ELSIF stRunPara.iPumpType=RudongPump_PumpType.V THEN
	stModbusAddress.iPumpType_Address:=1000;
	stModbusAddress.iHosePipeType_Address:=1001;	
	stModbusAddress.iFluVolumeSet_Address:=1015;
	stModbusAddress.iRuntimeSet_Address:=1018;
	stModbusAddress.iIntervalTime_Address:=1021;
	stModbusAddress.iCycleNumber_Address:=1023;
	stModbusAddress.iBackAngle_Address:=1007;
	stModbusAddress.iMoveDirection_Address:=1009;
	stModbusAddress.iStartStop_Address:=1008;
	stModbusAddress.iFullSpeedStartStop_Address:=1010;
	stModbusAddress.iModuleAddress_Address:=0;//等于0表示不写入
	stModbusAddress.iModuleStartStop_Address:=2003;
	stModbusAddress.iModuleRealFluVolumeSet_Address:=2004;
	stModbusAddress.iRecoveryCalCoefficient_Address:=2006;

	
	
END_IF
END_ACTION

ACTION ACT_PumpPar:
//
(*************************检测配置参数是否匹配成功*********************************)
IF stRunPara.iPumpType=RudongPump_PumpType.DFPluse THEN
	//MiniPump泵头
	IF  stRunPara.iPumpTypeSet=RudongPump_PumpHeadType.MiniPump01 THEN
		st_IOData.O_PumpType:=0;//泵头值为0
			IF stRunPara.iHosePipeTypeSet=RudongPump_SoftPipeType.P13 THEN//13#软管
				st_IOData.O_HosePipeType:=13;//软管类型值13
				IF rFluVolumeSet*1000/135<0.1 THEN
					iMinRunTime:=	0.1;
				ELSE
					iMinRunTime:=	(rFluVolumeSet*1000/135)*0.2+iMinRunTime;
				END_IF
				iMaxRunTime:=	rFluVolumeSet/0.45;//最大流量(0.45微升/秒,0.0024ml/min)	
			ELSIF stRunPara.iHosePipeTypeSet=RudongPump_SoftPipeType.P14 THEN//14#软管
				st_IOData.O_HosePipeType:=14;
				IF rFluVolumeSet*1000/570<0.1 THEN
					iMinRunTime:=	0.1;
				ELSE
					iMinRunTime:=	rFluVolumeSet*1000/135;
				END_IF
				iMaxRunTime:=	(rFluVolumeSet/1.9)*0.2+iMinRunTime;	
			ELSIF stRunPara.iHosePipeTypeSet=RudongPump_SoftPipeType.P19 THEN//19#软管
				st_IOData.O_HosePipeType:=19;
				IF rFluVolumeSet*1000/1240<0.1 THEN
					iMinRunTime:=	0.1;
				ELSE
					iMinRunTime:=	rFluVolumeSet*1000/1240;
				END_IF
				iMaxRunTime:=	(rFluVolumeSet*1000/4.13)*0.1+iMinRunTime;		
			ELSIF stRunPara.iHosePipeTypeSet=RudongPump_SoftPipeType.P16 THEN//16#软管
				st_IOData.O_HosePipeType:=16;
				IF rFluVolumeSet*1000/1880<0.1 THEN
					iMinRunTime:=	0.1;
				ELSE
					iMinRunTime:=	rFluVolumeSet*1000/1880;
				END_IF
				iMaxRunTime:=	(rFluVolumeSet*1000/6.28)*0.2+iMinRunTime;	
			ELSIF stRunPara.iHosePipeTypeSet=RudongPump_SoftPipeType.P25 THEN//25#软管
				st_IOData.O_HosePipeType:=25;
				IF rFluVolumeSet*1000/3100<0.1 THEN
					iMinRunTime:=	0.1;
				ELSE
					iMinRunTime:=	rFluVolumeSet*1000/3100;
				END_IF
				iMaxRunTime:=	(rFluVolumeSet*1000/10.33)*0.2+iMinRunTime;			
		ELSE
				eERRORID:=RudongPump_ERROR.FLT_CONFIGURE_PARA;		
		END_IF
	//UD15
	ELSIF  stRunPara.iPumpTypeSet=RudongPump_PumpHeadType.UD15 THEN
		st_IOData.O_PumpType:=1;//泵头值为0
			IF stRunPara.iHosePipeTypeSet=RudongPump_SoftPipeType.P16 THEN//16#软管
				st_IOData.O_HosePipeType:=16;
				IF rFluVolumeSet*1000/4000<0.1 THEN
					iMinRunTime:=	0.1;
				ELSE
					iMinRunTime:=	rFluVolumeSet*1000/4000;
				END_IF
				iMaxRunTime:=	(rFluVolumeSet*1000/13.33)*0.2+iMinRunTime;		
			ELSIF stRunPara.iHosePipeTypeSet=RudongPump_SoftPipeType.P17 THEN//17#软管
				st_IOData.O_HosePipeType:=17;
				IF rFluVolumeSet*1000/15000<0.1 THEN
					iMinRunTime:=	0.1;
				ELSE
					iMinRunTime:=	rFluVolumeSet*1000/15000;
				END_IF
				iMaxRunTime:=	(rFluVolumeSet*1000/50)*0.2+iMinRunTime;	
			ELSIF stRunPara.iHosePipeTypeSet=RudongPump_SoftPipeType.P25 THEN//25#软管
				st_IOData.O_HosePipeType:=25;
				IF rFluVolumeSet*1000/8000<0.1 THEN
					iMinRunTime:=	0.1;
				ELSE
					iMinRunTime:=	rFluVolumeSet*1000/8000;
				END_IF
				iMaxRunTime:=	(rFluVolumeSet*1000/26.66)*0.2+iMinRunTime;			
		ELSE
				eERRORID:=RudongPump_ERROR.FLT_CONFIGURE_PARA;		
		END_IF

	END_IF
ELSE
		eERRORID:=RudongPump_ERROR.FLT_CONFIGURE_PARA;
END_IF


(*
//MiniPump01泵头
IF  stRunPara.iPumpTypeSet=RudongPump_PumpHeadType.MiniPump01 THEN
		IF stRunPara.iHosePipeTypeSet=RudongPump_SoftPipeType.P13 THEN//13#软管
			iMinRunTime:=	(rFluVolumeSet/8)*60;//最大流量(135微升/秒,8.28ml/min)
			iMaxRunTime:=	(rFluVolumeSet/0.45)*60;//最大流量(0.45微升/秒,0.0024ml/min)	
		ELSIF stRunPara.iHosePipeTypeSet=RudongPump_SoftPipeType.P14 THEN//14#软管
			iMinRunTime:=	(rFluVolumeSet/33)*60;
			iMaxRunTime:=	(rFluVolumeSet/1.9)*60;
		ELSIF stRunPara.iHosePipeTypeSet=RudongPump_SoftPipeType.P19 THEN//19#软管
			iMinRunTime:=	(rFluVolumeSet/77)*60;
			iMaxRunTime:=	(rFluVolumeSet/4.13)*60;	
		ELSIF stRunPara.iHosePipeTypeSet=RudongPump_SoftPipeType.P16 THEN//16#软管
			iMinRunTime:=	(rFluVolumeSet/114)*60;
			iMaxRunTime:=	(rFluVolumeSet/6.28)*60;	
		ELSIF stRunPara.iHosePipeTypeSet=RudongPump_SoftPipeType.P25 THEN//25#软管
			iMinRunTime:=	(rFluVolumeSet/190)*60;
			iMaxRunTime:=	(rFluVolumeSet/10.33)*60;		
		ELSIF stRunPara.iHosePipeTypeSet=RudongPump_SoftPipeType.P1_1 THEN//1x1#软管
			iMinRunTime:=	(rFluVolumeSet/15)*60;
			iMaxRunTime:=	(rFluVolumeSet/4.5)*60;	
		ELSIF stRunPara.iHosePipeTypeSet=RudongPump_SoftPipeType.P2_1 THEN//2x1#软管
			iMinRunTime:=	(rFluVolumeSet/54)*60;
			iMaxRunTime:=	(rFluVolumeSet/4.5)*60;		
		ELSIF stRunPara.iHosePipeTypeSet=RudongPump_SoftPipeType.P2_5_1 THEN//2.5x1#软管
			iMinRunTime:=	(rFluVolumeSet/76)*60;
			iMaxRunTime:=	(rFluVolumeSet/5)*60;		
		ELSIF stRunPara.iHosePipeTypeSet=RudongPump_SoftPipeType.P3_1 THEN//3x1#软管
			iMinRunTime:=	(rFluVolumeSet/108)*60;
			iMaxRunTime:=	(rFluVolumeSet/5)*60;
	ELSE
			eERRORID:=RudongPump_ERROR.FLT_CONFIGURE_PARA;		
	END_IF		
	
//MiniPump02泵头
ELSIF  stRunPara.iPumpTypeSet=RudongPump_PumpHeadType.MiniPump02 THEN
	IF stRunPara.iHosePipeTypeSet=RudongPump_SoftPipeType.P1_1 THEN//1x1#软管
		iMinRunTime:=	(rFluVolumeSet/15.01)*60;
		iMaxRunTime:=	(rFluVolumeSet/0.005)*60;	
	ELSIF stRunPara.iHosePipeTypeSet=RudongPump_SoftPipeType.P2_1 THEN//2x1#软管
		iMinRunTime:=	(rFluVolumeSet/54.63)*60;
		iMaxRunTime:=	(rFluVolumeSet/0.018)*60;		
	ELSIF stRunPara.iHosePipeTypeSet=RudongPump_SoftPipeType.P2_5_1 THEN//2.5x1#软管
		iMinRunTime:=	(rFluVolumeSet/76.84)*60;
		iMaxRunTime:=	(rFluVolumeSet/0.0256)*60;
	ELSE
			eERRORID:=RudongPump_ERROR.FLT_CONFIGURE_PARA;						
	END_IF	

//HandyPump01泵头
ELSIF  stRunPara.iPumpTypeSet=RudongPump_PumpHeadType.HandyPump01 THEN
	IF stRunPara.iHosePipeTypeSet=RudongPump_SoftPipeType.P13 THEN//13#软管,三滚轮
		iMinRunTime:=	(rFluVolumeSet/10)*60;
		iMaxRunTime:=	(rFluVolumeSet/0.0033)*60;	
	ELSIF stRunPara.iHosePipeTypeSet=RudongPump_SoftPipeType.P14 THEN//14#软管,三滚轮
		iMinRunTime:=	(rFluVolumeSet/56)*60;
		iMaxRunTime:=	(rFluVolumeSet/0.0187)*60;		
	ELSIF stRunPara.iHosePipeTypeSet=RudongPump_SoftPipeType.P19 THEN//19#软管,三滚轮
		iMinRunTime:=	(rFluVolumeSet/111)*60;
		iMaxRunTime:=	(rFluVolumeSet/0.0371)*60;
	ELSIF stRunPara.iHosePipeTypeSet=RudongPump_SoftPipeType.P16 THEN//16#软管,三滚轮
		iMinRunTime:=	(rFluVolumeSet/190)*60;
		iMaxRunTime:=	(rFluVolumeSet/0.0636)*60;		
	ELSIF stRunPara.iHosePipeTypeSet=RudongPump_SoftPipeType.P25 THEN//25#软管,三滚轮
		iMinRunTime:=	(rFluVolumeSet/365)*60;
		iMaxRunTime:=	(rFluVolumeSet/0.1219)*60;
	ELSE
			eERRORID:=RudongPump_ERROR.FLT_CONFIGURE_PARA;						
	END_IF

//HandyPump02泵头
ELSIF  stRunPara.iPumpTypeSet=RudongPump_PumpHeadType.HandyPump02 THEN
	IF stRunPara.iHosePipeTypeSet=RudongPump_SoftPipeType.P13 THEN//13#软管,三滚轮
		iMinRunTime:=	(rFluVolumeSet/10)*60;
		iMaxRunTime:=	(rFluVolumeSet/0.0033)*60;	
	ELSIF stRunPara.iHosePipeTypeSet=RudongPump_SoftPipeType.P14 THEN//14#软管,三滚轮
		iMinRunTime:=	(rFluVolumeSet/56)*60;
		iMaxRunTime:=	(rFluVolumeSet/0.0187)*60;		
	ELSIF stRunPara.iHosePipeTypeSet=RudongPump_SoftPipeType.P19 THEN//19#软管,三滚轮
		iMinRunTime:=	(rFluVolumeSet/111)*60;
		iMaxRunTime:=	(rFluVolumeSet/0.0371)*60;
	ELSIF stRunPara.iHosePipeTypeSet=RudongPump_SoftPipeType.P16 THEN//16#软管,三滚轮
		iMinRunTime:=	(rFluVolumeSet/190)*60;
		iMaxRunTime:=	(rFluVolumeSet/0.0636)*60;	
	ELSE
			eERRORID:=RudongPump_ERROR.FLT_CONFIGURE_PARA;							
	END_IF

//EasyPumpI_III泵头,单通道
ELSIF  stRunPara.iPumpTypeSet=RudongPump_PumpHeadType.EasyPumpI_III THEN
	IF stRunPara.iHosePipeTypeSet=RudongPump_SoftPipeType.P13 THEN//13#软管
		iMinRunTime:=	(rFluVolumeSet/32)*60;
		iMaxRunTime:=	(rFluVolumeSet/0.0053)*60;	
	ELSIF stRunPara.iHosePipeTypeSet=RudongPump_SoftPipeType.P14 THEN//14#软管
		iMinRunTime:=	(rFluVolumeSet/162)*60;
		iMaxRunTime:=	(rFluVolumeSet/0.027)*60;		
	ELSIF stRunPara.iHosePipeTypeSet=RudongPump_SoftPipeType.P19 THEN//19#软管
		iMinRunTime:=	(rFluVolumeSet/330)*60;
		iMaxRunTime:=	(rFluVolumeSet/0.055)*60;
	ELSIF stRunPara.iHosePipeTypeSet=RudongPump_SoftPipeType.P16 THEN//16#软管
		iMinRunTime:=	(rFluVolumeSet/560)*60;
		iMaxRunTime:=	(rFluVolumeSet/0.093)*60;	
	ELSIF stRunPara.iHosePipeTypeSet=RudongPump_SoftPipeType.P25 THEN//25#软管
		iMinRunTime:=	(rFluVolumeSet/1180)*60;
		iMaxRunTime:=	(rFluVolumeSet/0.197)*60;	
	ELSIF stRunPara.iHosePipeTypeSet=RudongPump_SoftPipeType.P17 THEN//17#软管
		iMinRunTime:=	(rFluVolumeSet/2000)*60;
		iMaxRunTime:=	(rFluVolumeSet/0.333)*60;	
	ELSIF stRunPara.iHosePipeTypeSet=RudongPump_SoftPipeType.P18 THEN//18#软管
		iMinRunTime:=	(rFluVolumeSet/2580)*60;
		iMaxRunTime:=	(rFluVolumeSet/0.430)*60;	
	ELSE
			eERRORID:=RudongPump_ERROR.FLT_CONFIGURE_PARA;							
	END_IF

//EasyPumpII_IV泵头,单通道
ELSIF  stRunPara.iPumpTypeSet=RudongPump_PumpHeadType.EasyPumpII_IV THEN
	IF stRunPara.iHosePipeTypeSet=RudongPump_SoftPipeType.P15 THEN//15#软管
		iMinRunTime:=	(rFluVolumeSet/1080)*60;
		iMaxRunTime:=	(rFluVolumeSet/0.0180)*60;	
	ELSIF stRunPara.iHosePipeTypeSet=RudongPump_SoftPipeType.P24 THEN//24#软管
		iMinRunTime:=	(rFluVolumeSet/1640)*60;
		iMaxRunTime:=	(rFluVolumeSet/0.273)*60;		
	ELSIF stRunPara.iHosePipeTypeSet=RudongPump_SoftPipeType.P35 THEN//35#软管
		iMinRunTime:=	(rFluVolumeSet/2300)*60;
		iMaxRunTime:=	(rFluVolumeSet/0.383)*60;
	ELSIF stRunPara.iHosePipeTypeSet=RudongPump_SoftPipeType.P36 THEN//36#软管
		iMinRunTime:=	(rFluVolumeSet/3100)*60;
		iMaxRunTime:=	(rFluVolumeSet/0.517)*60;	
	ELSE
			eERRORID:=RudongPump_ERROR.FLT_CONFIGURE_PARA;							
	END_IF

//EasyPumpV_VI泵头,双通道
ELSIF  stRunPara.iPumpTypeSet=RudongPump_PumpHeadType.EasyPumpV_VI THEN
		IF stRunPara.iHosePipeTypeSet=RudongPump_SoftPipeType.P13 THEN//13#软管
		iMinRunTime:=	(rFluVolumeSet/32)*60;
		iMaxRunTime:=	(rFluVolumeSet/0.0053)*60;	
	ELSIF stRunPara.iHosePipeTypeSet=RudongPump_SoftPipeType.P14 THEN//14#软管
		iMinRunTime:=	(rFluVolumeSet/162)*60;
		iMaxRunTime:=	(rFluVolumeSet/0.0027)*60;		
	ELSIF stRunPara.iHosePipeTypeSet=RudongPump_SoftPipeType.P19 THEN//19#软管
		iMinRunTime:=	(rFluVolumeSet/330)*60;
		iMaxRunTime:=	(rFluVolumeSet/0.0055)*60;
	ELSIF stRunPara.iHosePipeTypeSet=RudongPump_SoftPipeType.P16 THEN//16#软管
		iMinRunTime:=	(rFluVolumeSet/560)*60;
		iMaxRunTime:=	(rFluVolumeSet/0.093)*60;		
	ELSIF stRunPara.iHosePipeTypeSet=RudongPump_SoftPipeType.P25 THEN//25#软管
		iMinRunTime:=	(rFluVolumeSet/1180)*60;
		iMaxRunTime:=	(rFluVolumeSet/0.197)*60;
	ELSE
			eERRORID:=RudongPump_ERROR.FLT_CONFIGURE_PARA;							
	END_IF
	
END_IF


END_IF

*)
		


//参数超出范围报错	
IF rFluVolumeSet<>0 THEN
	IF rRuntimeSet<iMinRunTime OR rRuntimeSet>iMaxRunTime OR  iMaxRunTime<iMinRunTime THEN
		eERRORID:=RudongPump_ERROR.FLT_CONFIGURE_PARA;
	END_IF
END_IF
END_ACTION

ACTION ACTMap:
ACT_GetModbusAddress();
_fResetCheck(CLK:=xResetRequest);
xRdyCmd := eState = STATE.DORMANT AND eERRORID = RudongPump_ERROR.No_ERROR;//检测是否允许指令控制(初始状态，没有报警发生)
xDone:=_xDone AND xExecute;
xError:=eState=STATE.INERROR;//报错发生
(**********************************检测是否有模式切换********************************)
_rManual(CLK:=xAutoMode);
_fManual(CLK:=xAutoMode);
IF eState <> STATE.DORMANT//只有在运行的时候，才会检测是否有模式切换发生
THEN
	IF _rManual.Q OR _fManual.Q
	THEN
		_xModeChange := TRUE;//通知系统有模式切换发生
	END_IF	
END_IF
IF eState = STATE.DORMANT//要是待机模式下，切换模式，是不会起作用的
THEN
	_xModeChange := FALSE;
END_IF


////
//调用MODBUS TCP功能
_fbModbusTCP.stSysPar.sRemoteHost:=stPara.strSlaveIP;//'192.168.1.20';
_fbModbusTCP.stSysPar.nRemotePort:=stPara.nRemotePort;
_fbModbusTCP.stSysPar.xSlaveAdr:=stPara.bySlaveID;
_fbModbusTCP(
	stParIn:= , 
	stSysPar:= , 
	xResetRequest:=xResetRequest , 
	stOpera:= , 
	xDone=> , 
	xBusy=> , 
	xError=> , 
	eERRORID=> , 
	eTCPErrorID=> , 	
	sModbusError=> , 
	xRdyCmd=> , 
	sError=> , 
	stParOut=> );
END_ACTION

METHOD PROTECTED CmdCalParWrite
VAR_OUTPUT
	xComplete: BOOL;
END_VAR
// return the real actual fault number
IF eERRORID <> RudongPump_ERROR.No_ERROR
THEN
  RETURN;  
END_IF

CASE _diCmdState OF	

	0://清空缓冲区
		SysMemSet(ADR(_fbModbusTCP.stParIn.aSendBuffer),0,SIZEOF(_fbModbusTCP.stParIn.aSendBuffer));		
		IF _fbModbusTCP.xRdyCmd THEN
			_diCmdState:=_diCmdState+1;
		ELSE
			eERRORID:=RudongPump_ERROR.FLT_Mobdus;
			_diCmdState:=999;
		END_IF
		
	1://单元实际液量设定
		_fbModbusTCP.stParIn.iHoldingRegisterAddress:=stModbusAddress.iModuleRealFluVolumeSet_Address;
		_fbModbusTCP.stParIn.iHoldingRegisterNum:=2;	
		_pDataControl:=ADR(iModuleRealVolume);	
 		_fbModbusTCP.stParIn.aSendBuffer[1]:=	_pDataControl[3];
 		_fbModbusTCP.stParIn.aSendBuffer[2]:=	_pDataControl[2];		
 		_fbModbusTCP.stParIn.aSendBuffer[3]:=	_pDataControl[1];		
 		_fbModbusTCP.stParIn.aSendBuffer[4]:=	_pDataControl[0];		
		_fbModbusTCP.stOpera.xSetMultiHoldingRegister:=TRUE;
		IF _fbModbusTCP.xDone THEN
			_fbModbusTCP.xExecute:=FALSE;
			_diCmdState:=_diCmdState+1;
		END_IF
		IF _fbModbusTCP.xError THEN
			eERRORID:=RudongPump_ERROR.FLT_Mobdus;
			_diCmdState:=999;
		END_IF
		
	2://
		xComplete := TRUE; 
		
	ELSE
		;	
END_CASE
END_METHOD

METHOD PROTECTED CmdCalReset
VAR_OUTPUT
	xComplete: BOOL;
END_VAR
// return the real actual fault number
IF eERRORID <> RudongPump_ERROR.No_ERROR
THEN
  RETURN;  
END_IF

CASE _diCmdState OF	
		
	0://清空缓冲区
		SysMemSet(ADR(_fbModbusTCP.stParIn.aSendBuffer),0,SIZEOF(_fbModbusTCP.stParIn.aSendBuffer));		
		IF _fbModbusTCP.xRdyCmd THEN
			_diCmdState:=_diCmdState+1;
		ELSE
			eERRORID:=RudongPump_ERROR.FLT_Mobdus;
			_diCmdState:=999;
		END_IF
		
	1://发送灌装系数复位指令
 		_fbModbusTCP.stParIn.aSendBuffer[1]:=16#00;
 		_fbModbusTCP.stParIn.aSendBuffer[2]:=16#01;		
		_fbModbusTCP.stParIn.iHoldingRegisterAddress:=stModbusAddress.iRecoveryCalCoefficient_Address;
		_fbModbusTCP.stParIn.iHoldingRegisterNum:=1;		 	
		_fbModbusTCP.stOpera.xSetSingalHoldingRegister:=TRUE;
		IF _fbModbusTCP.xDone THEN
			_fbModbusTCP.xExecute:=FALSE;
			_diCmdState:=_diCmdState+1;
		END_IF
		IF _fbModbusTCP.xError THEN
			eERRORID:=RudongPump_ERROR.FLT_Mobdus;
			_diCmdState:=999;
		END_IF

	2://
		xComplete := TRUE; 
		
	ELSE
		;	
END_CASE
END_METHOD

METHOD PROTECTED CmdPumpCal
VAR_OUTPUT
	xComplete: BOOL;
END_VAR
// return the real actual fault number
IF eERRORID <> RudongPump_ERROR.No_ERROR
THEN
  RETURN;  
END_IF

CASE _diCmdState OF	
	0://清空缓冲区
		SysMemSet(ADR(_fbModbusTCP.stParIn.aSendBuffer),0,SIZEOF(_fbModbusTCP.stParIn.aSendBuffer));		
		IF _fbModbusTCP.xRdyCmd THEN
			_diCmdState:=_diCmdState+1;
		ELSE
			eERRORID:=RudongPump_ERROR.FLT_Mobdus;
			_diCmdState:=999;
		END_IF
	
	 1://发送灌装液量,1002,REAL
		_fbModbusTCP.stParIn.iHoldingRegisterAddress:=stModbusAddress.iFluVolumeSet_Address;
		_fbModbusTCP.stParIn.iHoldingRegisterNum:=2;	
		_pDataControl:=ADR(rFluVolumeSet);	
 		_fbModbusTCP.stParIn.aSendBuffer[1]:=	_pDataControl[3];
 		_fbModbusTCP.stParIn.aSendBuffer[2]:=	_pDataControl[2];		
 		_fbModbusTCP.stParIn.aSendBuffer[3]:=	_pDataControl[1];		
 		_fbModbusTCP.stParIn.aSendBuffer[4]:=	_pDataControl[0];		
		_fbModbusTCP.stOpera.xSetMultiHoldingRegister:=TRUE;
		IF _fbModbusTCP.xDone THEN
			_fbModbusTCP.xExecute:=FALSE;
			_diCmdState:=_diCmdState+1;
		END_IF
		IF _fbModbusTCP.xError THEN
			eERRORID:=RudongPump_ERROR.FLT_Mobdus;
			_diCmdState:=999;
		END_IF		
	
	 2://发送灌装时间,1004,REAL
		_fbModbusTCP.stParIn.iHoldingRegisterAddress:=stModbusAddress.iRuntimeSet_Address;
		_fbModbusTCP.stParIn.iHoldingRegisterNum:=2;
		rRuntimeSet			:=stRunPara.rCalTime;
		_pDataControl:=ADR(rRuntimeSet);	
 		_fbModbusTCP.stParIn.aSendBuffer[1]:=	_pDataControl[3];
 		_fbModbusTCP.stParIn.aSendBuffer[2]:=	_pDataControl[2];		
 		_fbModbusTCP.stParIn.aSendBuffer[3]:=	_pDataControl[1];		
 		_fbModbusTCP.stParIn.aSendBuffer[4]:=	_pDataControl[0];		
		_fbModbusTCP.stOpera.xSetMultiHoldingRegister:=TRUE;
		IF _fbModbusTCP.xDone THEN
			_fbModbusTCP.xExecute:=FALSE;
			_diCmdState:=_diCmdState+1;
		END_IF
		IF _fbModbusTCP.xError THEN
			eERRORID:=RudongPump_ERROR.FLT_Mobdus;
			_diCmdState:=999;
		END_IF

	 3://发送灌装方向,1010,UINT
		IF eCmd = RudongPump_CMD.Cmd_Push OR eCmd = RudongPump_CMD.Cmd_CalPump
		THEN
			_fbModbusTCP.stParIn.aSendBuffer[1]:=16#00;
			_fbModbusTCP.stParIn.aSendBuffer[2]:=16#01;		
		END_IF
		IF eCmd = RudongPump_CMD.Cmd_Pull 
		THEN
			_fbModbusTCP.stParIn.aSendBuffer[1]:=16#00;
			_fbModbusTCP.stParIn.aSendBuffer[2]:=16#00;			
		END_IF		
		_fbModbusTCP.stParIn.iHoldingRegisterAddress:=stModbusAddress.iMoveDirection_Address;
		_fbModbusTCP.stParIn.iHoldingRegisterNum:=1;			 	
		_fbModbusTCP.stOpera.xSetSingalHoldingRegister:=TRUE;
		IF _fbModbusTCP.xDone THEN
			_fbModbusTCP.xExecute:=FALSE;
			_diCmdState:=_diCmdState+1;
		END_IF
		IF _fbModbusTCP.xError THEN
			eERRORID:=RudongPump_ERROR.FLT_Mobdus;
			_diCmdState:=999;
		END_IF		

	4://发送重复次数,1008,UINT
		_pDataControl:=ADR(iCycleNumber);	
 		_fbModbusTCP.stParIn.aSendBuffer[1]:=_pDataControl[1];
 		_fbModbusTCP.stParIn.aSendBuffer[2]:=_pDataControl[0];		
		_fbModbusTCP.stParIn.iHoldingRegisterAddress:=stModbusAddress.iCycleNumber_Address;
		_fbModbusTCP.stParIn.iHoldingRegisterNum:=1;		 	
		_fbModbusTCP.stOpera.xSetSingalHoldingRegister:=TRUE;
		IF _fbModbusTCP.xDone THEN
			_fbModbusTCP.xExecute:=FALSE;
			_diCmdState:=_diCmdState+1;
		END_IF
		IF _fbModbusTCP.xError THEN
			eERRORID:=RudongPump_ERROR.FLT_Mobdus;
			_diCmdState:=999;
		END_IF	
		
	5://单元地址设定,2000,UINT
		_pDataControl:=ADR(iModuleAdress);	
 		_fbModbusTCP.stParIn.aSendBuffer[1]:=_pDataControl[1];
 		_fbModbusTCP.stParIn.aSendBuffer[2]:=_pDataControl[0];		
		_fbModbusTCP.stParIn.iHoldingRegisterAddress:=stModbusAddress.iModuleAddress_Address;
		_fbModbusTCP.stParIn.iHoldingRegisterNum:=1;		
		IF  _fbModbusTCP.stParIn.iHoldingRegisterAddress<>0 THEN	
			_fbModbusTCP.stOpera.xSetSingalHoldingRegister:=TRUE;
			IF _fbModbusTCP.xDone THEN
				_fbModbusTCP.xExecute:=FALSE;
				_diCmdState:=_diCmdState+1;
			END_IF
			IF _fbModbusTCP.xError THEN
				eERRORID:=RudongPump_ERROR.FLT_Mobdus;
				_diCmdState:=999;
			END_IF
		ELSE
			_diCmdState:=_diCmdState+1;//地址为0 则跳过设置
		END_IF
		
	6://灌装启动,2003,UINT	
 		_fbModbusTCP.stParIn.aSendBuffer[1]:=16#00;
 		_fbModbusTCP.stParIn.aSendBuffer[2]:=16#01;		
		_fbModbusTCP.stParIn.iHoldingRegisterAddress:=stModbusAddress.iModuleStartStop_Address;
		_fbModbusTCP.stParIn.iHoldingRegisterNum:=1;		 	
		_fbModbusTCP.stOpera.xSetSingalHoldingRegister:=TRUE;
		IF _fbModbusTCP.xDone THEN
			_fbModbusTCP.xExecute:=FALSE;
			_diCmdState:=_diCmdState+1;
		END_IF
		IF _fbModbusTCP.xError THEN
			eERRORID:=RudongPump_ERROR.FLT_Mobdus;
			_diCmdState:=999;
		END_IF

	7://查询蠕动泵运行状态,2003,UINT
		_fbModbusTCP.stParIn.iHoldingRegisterAddress:=stModbusAddress.iModuleStartStop_Address;
		_fbModbusTCP.stParIn.iHoldingRegisterNum:=1;		 	
		_fbModbusTCP.stOpera.xReadHoldingRegisters:=TRUE;
		IF _fbModbusTCP.xDone THEN
			_fbModbusTCP.xExecute:=FALSE;
			_diCmdState:=_diCmdState+1;
		END_IF
		IF _fbModbusTCP.xError THEN
			eERRORID:=RudongPump_ERROR.FLT_Mobdus;
			_diCmdState:=999;
		END_IF			
		
	8://判断运行状态,并延时
		IF _fbModbusTCP.stParOut.aRcvBuffer[1]=0 AND _fbModbusTCP.stParOut.aRcvBuffer[2]=0 THEN
			xComplete:=TRUE;
		ELSE
			xRunning:=TRUE;
			_tonDelay(IN:=TRUE,PT:=T#0.5S);
			IF _tonDelay.Q THEN
				_tonDelay(IN:=FALSE);
				_diCmdState:=7;
			END_IF
		END_IF
		
	ELSE
		;	
END_CASE
END_METHOD

METHOD PROTECTED CmdRunAction
VAR_OUTPUT
	xComplete: BOOL;
END_VAR
// return the real actual fault number
IF eERRORID <> RudongPump_ERROR.No_ERROR
THEN
  RETURN;  
END_IF

CASE _diCmdState OF	
	0://清空缓冲区
		SysMemSet(ADR(_fbModbusTCP.stParIn.aSendBuffer),0,SIZEOF(_fbModbusTCP.stParIn.aSendBuffer));		
		IF _fbModbusTCP.xRdyCmd THEN
			IF xNeedConfigurePara THEN
				_diCmdState:=_diCmdState+1;
			ELSE
				_diCmdState:=6;//如果不需要配置则直接启动
			END_IF			
		ELSE
			eERRORID:=RudongPump_ERROR.FLT_Mobdus;
			_diCmdState:=999;
		END_IF

	 1://发送虚假灌装时间,1004,REAL
		_fbModbusTCP.stParIn.iHoldingRegisterAddress:=stModbusAddress.iRuntimeSet_Address;
		_fbModbusTCP.stParIn.iHoldingRegisterNum:=2;
		_pDataControl:=ADR(iMaxRunTime);	
 		_fbModbusTCP.stParIn.aSendBuffer[1]:=	_pDataControl[3];
 		_fbModbusTCP.stParIn.aSendBuffer[2]:=	_pDataControl[2];		
 		_fbModbusTCP.stParIn.aSendBuffer[3]:=	_pDataControl[1];		
 		_fbModbusTCP.stParIn.aSendBuffer[4]:=	_pDataControl[0];		
		_fbModbusTCP.stOpera.xSetMultiHoldingRegister:=TRUE;
		IF _fbModbusTCP.xDone THEN
			_fbModbusTCP.xExecute:=FALSE;
			_diCmdState:=_diCmdState+1;
		END_IF
		IF _fbModbusTCP.xError THEN
			eERRORID:=RudongPump_ERROR.FLT_Mobdus;
			_diCmdState:=999;
		END_IF		
		
	 2://发送灌装液量,1002,REAL
		_fbModbusTCP.stParIn.iHoldingRegisterAddress:=stModbusAddress.iFluVolumeSet_Address;
		_fbModbusTCP.stParIn.iHoldingRegisterNum:=2;	
		_pDataControl:=ADR(rFluVolumeSet);	
 		_fbModbusTCP.stParIn.aSendBuffer[1]:=	_pDataControl[3];
 		_fbModbusTCP.stParIn.aSendBuffer[2]:=	_pDataControl[2];		
 		_fbModbusTCP.stParIn.aSendBuffer[3]:=	_pDataControl[1];		
 		_fbModbusTCP.stParIn.aSendBuffer[4]:=	_pDataControl[0];		
		_fbModbusTCP.stOpera.xSetMultiHoldingRegister:=TRUE;
		IF _fbModbusTCP.xDone THEN
			_fbModbusTCP.xExecute:=FALSE;
			_diCmdState:=_diCmdState+1;
		END_IF
		IF _fbModbusTCP.xError THEN
			eERRORID:=RudongPump_ERROR.FLT_Mobdus;
			_diCmdState:=999;
		END_IF			

	 3://发送实际灌装时间,1004,REAL
		_fbModbusTCP.stParIn.iHoldingRegisterAddress:=stModbusAddress.iRuntimeSet_Address;
		_fbModbusTCP.stParIn.iHoldingRegisterNum:=2;
		_pDataControl:=ADR(rRuntimeSet);	
 		_fbModbusTCP.stParIn.aSendBuffer[1]:=	_pDataControl[3];
 		_fbModbusTCP.stParIn.aSendBuffer[2]:=	_pDataControl[2];		
 		_fbModbusTCP.stParIn.aSendBuffer[3]:=	_pDataControl[1];		
 		_fbModbusTCP.stParIn.aSendBuffer[4]:=	_pDataControl[0];		
		_fbModbusTCP.stOpera.xSetMultiHoldingRegister:=TRUE;
		IF _fbModbusTCP.xDone THEN
			_fbModbusTCP.xExecute:=FALSE;
			_diCmdState:=_diCmdState+1;
		END_IF
		IF _fbModbusTCP.xError THEN
			eERRORID:=RudongPump_ERROR.FLT_Mobdus;
			_diCmdState:=999;
		END_IF
		
	 4://发送灌装方向,1010,UINT
		IF eCmd = RudongPump_CMD.Cmd_Push
		THEN
			_fbModbusTCP.stParIn.aSendBuffer[1]:=16#00;
			_fbModbusTCP.stParIn.aSendBuffer[2]:=16#01;		
		END_IF
		IF eCmd = RudongPump_CMD.Cmd_Pull 
		THEN
			_fbModbusTCP.stParIn.aSendBuffer[1]:=16#00;
			_fbModbusTCP.stParIn.aSendBuffer[2]:=16#00;			
		END_IF		
		_fbModbusTCP.stParIn.iHoldingRegisterAddress:=stModbusAddress.iMoveDirection_Address;
		_fbModbusTCP.stParIn.iHoldingRegisterNum:=1;			 	
		_fbModbusTCP.stOpera.xSetSingalHoldingRegister:=TRUE;
		IF _fbModbusTCP.xDone THEN
			_fbModbusTCP.xExecute:=FALSE;
			_diCmdState:=_diCmdState+1;
		END_IF
		IF _fbModbusTCP.xError THEN
			eERRORID:=RudongPump_ERROR.FLT_Mobdus;
			_diCmdState:=999;
		END_IF		

	5://发送重复次数,1008,UINT
		_pDataControl:=ADR(iCycleNumber);	
 		_fbModbusTCP.stParIn.aSendBuffer[1]:=_pDataControl[1];
 		_fbModbusTCP.stParIn.aSendBuffer[2]:=_pDataControl[0];		
		_fbModbusTCP.stParIn.iHoldingRegisterAddress:=stModbusAddress.iCycleNumber_Address;
		_fbModbusTCP.stParIn.iHoldingRegisterNum:=1;		 	
		_fbModbusTCP.stOpera.xSetSingalHoldingRegister:=TRUE;
		IF _fbModbusTCP.xDone THEN
			_fbModbusTCP.xExecute:=FALSE;
			_diCmdState:=_diCmdState+1;
		END_IF
		IF _fbModbusTCP.xError THEN
			eERRORID:=RudongPump_ERROR.FLT_Mobdus;
			_diCmdState:=999;
		END_IF

	6://发送启动,1011,UINT
		_fbModbusTCP.stParIn.aSendBuffer[1]:=16#00;
		_fbModbusTCP.stParIn.aSendBuffer[2]:=16#01;	
		_fbModbusTCP.stParIn.iHoldingRegisterAddress:=stModbusAddress.iStartStop_Address;
		_fbModbusTCP.stParIn.iHoldingRegisterNum:=1;		 	
		_fbModbusTCP.stOpera.xSetSingalHoldingRegister:=TRUE;
		IF _fbModbusTCP.xDone THEN
			_fbModbusTCP.xExecute:=FALSE;
			_diCmdState:=_diCmdState+1;
		END_IF
		IF _fbModbusTCP.xError THEN
			eERRORID:=RudongPump_ERROR.FLT_Mobdus;
			_diCmdState:=999;
		END_IF
	7://查询蠕动泵运行状态,1011,UINT
		_fbModbusTCP.stParIn.iHoldingRegisterAddress:=stModbusAddress.iStartStop_Address;
		_fbModbusTCP.stParIn.iHoldingRegisterNum:=1;		 	
		_fbModbusTCP.stOpera.xReadHoldingRegisters:=TRUE;
		IF _fbModbusTCP.xDone THEN
			_fbModbusTCP.xExecute:=FALSE;
			_diCmdState:=_diCmdState+1;
		END_IF
		IF _fbModbusTCP.xError THEN
			eERRORID:=RudongPump_ERROR.FLT_Mobdus;
			_diCmdState:=999;
		END_IF			
		
	8://判断运行状态,并延时
		IF _fbModbusTCP.stParOut.aRcvBuffer[1]=0 AND _fbModbusTCP.stParOut.aRcvBuffer[2]=0 THEN
			xComplete:=TRUE;
		ELSE
			xRunning:=TRUE;
			_tonDelay(IN:=TRUE,PT:=T#1S);
			IF _tonDelay.Q THEN
				_tonDelay(IN:=FALSE);
				_diCmdState:=7;
			END_IF
		END_IF
	
	
		
	ELSE
		;	
END_CASE
END_METHOD

METHOD PROTECTED CyclicAction
VAR_OUTPUT
	xComplete: BOOL;
END_VAR
IF xAbort=0 THEN
    IF xFirstInvocation THEN
    (*
    * Staring
    * for then first (!) invocaion,
    * sample then input variables
    *)			
    _diCmdState:= 0;
		_iNGCount := 0;
		_iActRunNumber := 0;
		xFirstInvocation:=0;			
    END_IF    
    REPEAT 				
		  (**************************检查是否有硬件报错(检测总线是否报错)**********************************) 
			IF _xConnectError
			THEN
				eERRORID := RudongPump_ERROR.FLT_CONNECT;//子站通讯报警
			END_IF
		
	
			//检测停止指令是否发生
			_rStopCmdTrig(CLK:= NOT xEStop OR (stDeviceOpe.xStop_Hmi AND NOT xAutoMode AND NOT xDeviceRunning) OR (stDeviceOpe.xStop_Auto AND (xAutoMode OR xDeviceRunning))
													OR (stDeviceOpe.xFullSpeedStop_Hmi AND NOT xAutoMode AND NOT xDeviceRunning) OR (stDeviceOpe.xFullSpeedStop_Auto AND (xAutoMode OR xDeviceRunning)));		
		  IF _rStopCmdTrig.Q//检测到停止指令
			THEN
				_diCmdState := 0;
				eCmd := RudongPump_CMD.Cmd_Stop;
				_tonCmdTimeout(in:=FALSE);
				_tonDelay(IN:= FALSE);
				_tonTimeout(in:=FALSE);
			END_IF
			
			ACT_PumpPar();//检查参数	
			
			
			CASE eCmd OF//判断指令类型
				RudongPump_CMD.Cmd_Pull,RudongPump_CMD.Cmd_Push://执行夹爪指令(夹紧和松开指令)
					CmdRunAction(xComplete=> xComplete);	
							
				RudongPump_CMD.Cmd_Stop,RudongPump_CMD.Cmd_FullSpeedStop://执行过程中等待停止指令(分为运行停止和全速停止)
					mCmdStopAction(xComplete=> xComplete);
					
				RudongPump_CMD.Cmd_Configure://(用于配置参数)
					mCmdConfigureAction(xComplete=> xComplete);
					
				RudongPump_CMD.Cmd_FullSpeedPush,RudongPump_CMD.Cmd_FullSpeedPull://全速启动控制（用于清洗和充满试管）
					mCmdFullSpeedStartAction(xComplete=> xComplete);
					
				RudongPump_CMD.Cmd_CalPump:
					CmdPumpCal(xComplete=> xComplete);

				RudongPump_CMD.Cmd_CalReset:
					CmdCalReset(xComplete=> xComplete);		

				RudongPump_CMD.Cmd_CalParWrite:
					CmdCalParWrite(xComplete=> xComplete);		
				ELSE
					;	
				END_CASE		   
      UNTIL (TRUE)
	END_REPEAT
END_IF

IF xAbort OR xComplete OR eERRORID<>RudongPump_ERROR.No_ERROR THEN    
    (*
    * Cleaning
    * => free as much allocated resources as possible
    *)    
    tOperationTimer(IN:=0);
END_IF
END_METHOD

METHOD PRIVATE FINAL HandleAbortedState
VAR_INPUT
END_VAR
VAR_OUTPUT
	xAgain: BOOL;
END_VAR
VAR
	xComplete: BOOL;
END_VAR
IF xAborted AND xResetRequest THEN
    eState:=STATE.RESETING;
    xAgain:=1;
ELSE
    xBusy:=0;
    xAborted:=1;
    //xResetRequest:=(xExecute=0);
    xAgain:=0;(* !!! *)
END_IF
END_METHOD

METHOD PRIVATE FINAL HandleAbortingState
VAR_INPUT
END_VAR
VAR_OUTPUT
	xAgain: BOOL;
END_VAR
VAR
	xComplete: BOOL;
END_VAR
AbortAction(xComplete=> xComplete, eERRORID=> eERRORID);

IF eERRORID<>RudongPump_ERROR.No_ERROR THEN
    eState:=STATE.INERROR;
    xAgain:=1;
ELSIF xComplete THEN
    eState:=STATE.ABORTED;
    xAgain:=1;
END_IF
END_METHOD

METHOD PRIVATE FINAL HandleDoneState
VAR_INPUT
END_VAR
VAR_OUTPUT
	xAgain: BOOL;
END_VAR
//在运行过程中要是切换模式，再运行完成之后，检测到模式的切换，就需要回到初始位置，进行下一次执行准备
IF _xDone AND ((xExecute=0) OR ( _xModeChange AND NOT _xAutoOpe)  OR ( NOT xAutoMode AND NOT xDeviceRunning AND ( NOT _xAutoOpe OR _xHMIOpe))) THEN
	eState:=STATE.RESETING;
	xAgain:=1;
ELSE
	xBusy:=0;
	_xDone:=1;
	xAgain:=0;(* !!! *)
END_IF
END_METHOD

METHOD PRIVATE FINAL HandleDormantState
VAR_INPUT
END_VAR
VAR_OUTPUT
	xAgain: BOOL;
END_VAR
IF xExecute THEN
    xBusy:=1;
    eState:=STATE.EXECUTING;
    xAgain:=1;
END_IF
//下面两个报警一旦报警就需要发生
IF _xConnectError 
THEN//出现这个进行报警
	eERRORID := RudongPump_ERROR.FLT_CONNECT;//子站通讯报警
END_IF

IF _fResetCheck.Q//清空报警
THEN
	eERRORID := RudongPump_ERROR.No_ERROR;
END_IF
IF  xAutoMode OR xDeviceRunning THEN
	xAutomodeFlag:=TRUE;
ELSE
	xAutomodeFlag:=FALSE;
END_IF


IF eErrorID = RudongPump_ERROR.NO_ERROR 
THEN
	IF   xRunILC   THEN
		FOR k:=1 TO 5 BY 1 DO
			//PULL
			_rOperaTrig[k](CLK:=xRunILC AND (stDeviceOpe.xPull_Hmi[k] AND NOT xAutomodeFlag) OR (stDeviceOpe.xPull_Auto[k] AND xAutomodeFlag));
			IF _rOperaTrig[k].Q //
			THEN
				rFluVolumeSet	:=stRunPara.rPullFluVolume[k];
				rRuntimeSet		:=stRunPara.rPullRuntime[k];
				iCycleNumber	:=stRunPara.iPullCycleNumber[k];
				eCmd 			:= RudongPump_CMD.Cmd_Pull;
				xExecute		:= TRUE;
			END_IF		
			//PUSH
			_rOperaTrig[k+5](CLK:=xRunILC AND (stDeviceOpe.xPush_Hmi[k] AND NOT xAutomodeFlag) OR (stDeviceOpe.xPush_Auto[k] AND xAutomodeFlag));
			IF _rOperaTrig[k+5].Q 
			THEN
				rFluVolumeSet	:=stRunPara.rPushFluVolume[k];  
				rRuntimeSet		:=stRunPara.rPushRuntime[k];    
				iCycleNumber	:=stRunPara.iPushCycleNumber[k];
				eCmd 			:= RudongPump_CMD.Cmd_Push;
				xExecute 		:= TRUE;
			END_IF				
		END_FOR
		//STOP
		 IF(stDeviceOpe.xStop_Hmi AND  NOT xAutomodeFlag) OR NOT xEStop OR stDeviceOpe.xStop_Auto    THEN
				eCmd := RudongPump_CMD.Cmd_Stop;
				xExecute := TRUE;
		 END_IF
		//FullSpeedPull
		IF (stDeviceOpe.xFullSpeedPull_Hmi AND  NOT xAutomodeFlag) OR (stDeviceOpe.xFullSpeedPull_Auto AND  xAutomodeFlag) THEN
			eCmd := RudongPump_CMD.Cmd_FullSpeedPull;
			xExecute := TRUE;
		END_IF
		//FullSpeedPush
		IF (stDeviceOpe.xFullSpeedPush_Hmi AND NOT xAutomodeFlag ) OR (stDeviceOpe.xFullSpeedPush_Auto AND xAutomodeFlag) THEN	
			eCmd := RudongPump_CMD.Cmd_FullSpeedPush;
			xExecute := TRUE;
		END_IF
		//FullSpeedStop
		 IF (stDeviceOpe.xFullSpeedStop_Hmi AND NOT xAutomodeFlag) OR (stDeviceOpe.xFullSpeedStop_Auto AND xAutomodeFlag) THEN	
			eCmd := RudongPump_CMD.Cmd_FullSpeedStop;
			xExecute := TRUE;
		END_IF
		//Configure
		IF (stDeviceOpe.xConfigure_Hmi AND NOT xAutomodeFlag) OR (stDeviceOpe.xConfigure_Auto AND xAutomodeFlag) THEN	
			eCmd := RudongPump_CMD.Cmd_Configure;
			xExecute := TRUE;
		END_IF
		
	END_IF		
		//校准
		IF stDeviceOpe.xPumpCal_Hmi OR stDeviceOpe.xPumpCal_Auto THEN
			rFluVolumeSet		:=stRunPara.rCalFluVolume;
			rRuntimeSet			:=stRunPara.rCalTime;
			iCycleNumber		:=stRunPara.rCalNum;	
			iModuleAdress		:=stRunPara.iModuleAdress;
			iModuleSpeed		:=stRunPara.rModuleSpeed;		
			eCmd 				:= RudongPump_CMD.Cmd_CalPump;
			xExecute 			:= TRUE;		
		END_IF
		
		//复位校准系数为初始值
		IF stDeviceOpe.xResetCalcoeffCal_Hmi THEN	
			eCmd 				:= RudongPump_CMD.Cmd_CalReset;
			xExecute 			:= TRUE;		
		END_IF
	
		//校准参数写入
		IF stDeviceOpe.xCalParWrite_Hmi OR stDeviceOpe.xCalParWrite_Auto THEN	
			eCmd 								:= RudongPump_CMD.Cmd_CalParWrite;
			iModuleRealVolume		:=stRunPara.rModuleRealFluVolume;					
			xExecute 						:= TRUE;		
		END_IF	
			
END_IF
END_METHOD

METHOD PRIVATE FINAL  HandleErrorState
VAR_INPUT
END_VAR
VAR_OUTPUT
	xAgain: BOOL;
END_VAR
IF xRudongPump_ERROR AND  (xResetRequest OR NOT xExecute) THEN
    eState:=STATE.RESETING;
    xAgain:=1;
ELSE
    xBusy:=0;
    xRudongPump_ERROR:=1;    
    xAgain:=0;(* !!! *)
END_IF
END_METHOD

METHOD PRIVATE FINAL HandleExecutingState
VAR_INPUT
END_VAR
VAR_OUTPUT
	xAgain: BOOL;
END_VAR
VAR
	xComplete: BOOL;
END_VAR
IF xAbort=0 THEN   
    CyclicAction(xComplete=> xComplete);
END_IF

IF eERRORID<>RudongPump_ERROR.No_ERROR THEN
    eState:=STATE.INERROR;
    xAgain:=1;
ELSIF xAbort THEN
    eState:=STATE.ABORTING;
    xAgain:=1;
ELSIF xComplete THEN
    eState:=STATE.DONE;
    xAgain:=1;
END_IF
END_METHOD

METHOD PRIVATE FINAL HandleResettingState
VAR_INPUT
END_VAR
VAR_OUTPUT
	xAgain: BOOL;
END_VAR
VAR
	xComplete: BOOL;
END_VAR
ResetAction(xComplete=> xComplete);

IF xComplete THEN
	xExecute:=0;//清除输入指令 
    xBusy:=0;
    _xDone:=0;
    xRudongPump_ERROR:=0;
    xAborted:=0;
    eERRORID:=RudongPump_ERROR.No_ERROR;
    eState:=STATE.DORMANT;
    xFirstInvocation:=1;
    xAgain:=0;(* !!! *)
END_IF
END_METHOD

METHOD PROTECTED mCmdConfigureAction
VAR_OUTPUT
	xComplete: BOOL;
END_VAR
// return the real actual fault number
IF eERRORID <> RudongPump_ERROR.No_ERROR
THEN
  RETURN;  
END_IF

CASE _diCmdState OF

	0://清空缓冲区
		SysMemSet(ADR(_fbModbusTCP.stParIn.aSendBuffer),0,SIZEOF(_fbModbusTCP.stParIn.aSendBuffer));		
		IF _fbModbusTCP.xRdyCmd THEN
			_diCmdState:=_diCmdState+1;
		ELSE
			eERRORID:=RudongPump_ERROR.FLT_Mobdus;
			_diCmdState:=999;
		END_IF
		
	 1://发送泵头编号,1000,UINT
		_pDataControl:=ADR(st_IOData.O_PumpType);	
 		_fbModbusTCP.stParIn.aSendBuffer[1]:=_pDataControl[1];
 		_fbModbusTCP.stParIn.aSendBuffer[2]:=_pDataControl[0];		
		_fbModbusTCP.stParIn.iHoldingRegisterAddress:=stModbusAddress.iPumpType_Address;
		_fbModbusTCP.stParIn.iHoldingRegisterNum:=1;		 	
		_fbModbusTCP.stOpera.xSetSingalHoldingRegister:=TRUE;
		IF _fbModbusTCP.xDone THEN
			_fbModbusTCP.xExecute:=FALSE;
			_diCmdState:=_diCmdState+1;
		END_IF
		IF _fbModbusTCP.xError THEN
			eERRORID:=RudongPump_ERROR.FLT_Mobdus;
			_diCmdState:=999;
		END_IF

	 2://发送软管编号,1001,UINT
		_pDataControl:=ADR(st_IOData.O_HosePipeType);	
 		_fbModbusTCP.stParIn.aSendBuffer[1]:=_pDataControl[1];
 		_fbModbusTCP.stParIn.aSendBuffer[2]:=_pDataControl[0];		
		_fbModbusTCP.stParIn.iHoldingRegisterAddress:=stModbusAddress.iHosePipeType_Address;
		_fbModbusTCP.stParIn.iHoldingRegisterNum:=1;		 	
		_fbModbusTCP.stOpera.xSetSingalHoldingRegister:=TRUE;
		IF _fbModbusTCP.xDone THEN
			_fbModbusTCP.xExecute:=FALSE;
			_diCmdState:=_diCmdState+1;
		END_IF
		IF _fbModbusTCP.xError THEN
			eERRORID:=RudongPump_ERROR.FLT_Mobdus;
			_diCmdState:=999;
		END_IF

	3://
		xComplete:=TRUE;
















	ELSE
		;
END_CASE
END_METHOD

METHOD PROTECTED mCmdFullSpeedStartAction
VAR_OUTPUT
	xComplete: BOOL;
END_VAR
// return the real actual fault number
IF eERRORID <> RudongPump_ERROR.No_ERROR
THEN
  RETURN;  
END_IF

CASE _diCmdState OF
	0://清空缓冲区
		SysMemSet(ADR(_fbModbusTCP.stParIn.aSendBuffer),0,SIZEOF(_fbModbusTCP.stParIn.aSendBuffer));		
		IF _fbModbusTCP.xRdyCmd THEN
			_diCmdState:=_diCmdState+1;
		ELSE
			eERRORID:=RudongPump_ERROR.FLT_Mobdus;
			_diCmdState:=999;
		END_IF

	 1://发送灌装方向,1010,UINT
		IF eCmd = RudongPump_CMD.Cmd_FullSpeedPush
		THEN
			_fbModbusTCP.stParIn.aSendBuffer[1]:=16#00;
			_fbModbusTCP.stParIn.aSendBuffer[2]:=16#01;		
		END_IF
		IF eCmd = RudongPump_CMD.Cmd_FullSpeedPull 
		THEN
			_fbModbusTCP.stParIn.aSendBuffer[1]:=16#00;
			_fbModbusTCP.stParIn.aSendBuffer[2]:=16#00;			
		END_IF		
		_fbModbusTCP.stParIn.iHoldingRegisterAddress:=stModbusAddress.iMoveDirection_Address;
		_fbModbusTCP.stParIn.iHoldingRegisterNum:=1;			 	
		_fbModbusTCP.stOpera.xSetSingalHoldingRegister:=TRUE;
		IF _fbModbusTCP.xDone THEN
			_fbModbusTCP.xExecute:=FALSE;
			_diCmdState:=_diCmdState+1;
		END_IF
		IF _fbModbusTCP.xError THEN
			eERRORID:=RudongPump_ERROR.FLT_Mobdus;
			_diCmdState:=999;
		END_IF	
		
	2://发送启动,1012,UINT
		_fbModbusTCP.stParIn.aSendBuffer[1]:=16#00;
		_fbModbusTCP.stParIn.aSendBuffer[2]:=16#01;	
		_fbModbusTCP.stParIn.iHoldingRegisterAddress:=stModbusAddress.iFullSpeedStartStop_Address;
		_fbModbusTCP.stParIn.iHoldingRegisterNum:=1;		 	
		_fbModbusTCP.stOpera.xSetSingalHoldingRegister:=TRUE;
		IF _fbModbusTCP.xDone THEN
			_fbModbusTCP.xExecute:=FALSE;
			_diCmdState:=_diCmdState+1;
		END_IF
		IF _fbModbusTCP.xError THEN
			eERRORID:=RudongPump_ERROR.FLT_Mobdus;
			_diCmdState:=999;
		END_IF
		
	3://查询蠕动泵运行状态,1012,UINT
		_fbModbusTCP.stParIn.iHoldingRegisterAddress:=stModbusAddress.iStartStop_Address;
		_fbModbusTCP.stParIn.iHoldingRegisterNum:=1;		 	
		_fbModbusTCP.stOpera.xReadHoldingRegisters:=TRUE;
		IF _fbModbusTCP.xDone THEN
			_fbModbusTCP.xExecute:=FALSE;
			_diCmdState:=_diCmdState+1;
		END_IF
		IF _fbModbusTCP.xError THEN
			eERRORID:=RudongPump_ERROR.FLT_Mobdus;
			_diCmdState:=999;
		END_IF			
		
	4://判断运行状态,并延时
		IF _fbModbusTCP.stParOut.aRcvBuffer[1]<>0 OR _fbModbusTCP.stParOut.aRcvBuffer[2]<>0 THEN
			xRunning:=TRUE;
			xComplete:=TRUE;
		ELSE
			_tonDelay(IN:=TRUE,PT:=T#0.5S);
			IF _tonDelay.Q THEN
				_tonDelay(IN:=FALSE);
				_diCmdState:=2;
			END_IF
		END_IF		
		
		
	ELSE
		;
END_CASE
END_METHOD

METHOD PROTECTED mCmdStopAction
VAR_OUTPUT
	xComplete: BOOL;
END_VAR
// return the real actual fault number
IF eERRORID <> RudongPump_ERROR.No_ERROR
THEN
  RETURN;  
END_IF

CASE _diCmdState OF
	0://清空缓冲区
		_tonDelay(IN:=_fbModbusTCP.xRdyCmd,PT:=T#100MS);
		SysMemSet(ADR(_fbModbusTCP.stParIn.aSendBuffer),0,SIZEOF(_fbModbusTCP.stParIn.aSendBuffer));		
		IF _fbModbusTCP.xRdyCmd AND _tonDelay.Q THEN
			_diCmdState:=_diCmdState+1;
		ELSE
			_fbModbusTCP.xExecute:=FALSE;
		END_IF

	1://发送启动停止,1012,UINT
		_fbModbusTCP.stParIn.aSendBuffer[1]:=16#00;
		_fbModbusTCP.stParIn.aSendBuffer[2]:=16#00;	
		_fbModbusTCP.stParIn.iHoldingRegisterAddress:=stModbusAddress.iFullSpeedStartStop_Address;
		_fbModbusTCP.stParIn.iHoldingRegisterNum:=1;		 	
		_fbModbusTCP.stOpera.xSetSingalHoldingRegister:=TRUE;
		IF _fbModbusTCP.xDone THEN
			_fbModbusTCP.xExecute:=FALSE;
			_diCmdState:=_diCmdState+1;
		END_IF
		IF _fbModbusTCP.xError THEN
			eERRORID:=RudongPump_ERROR.FLT_Mobdus;
			_diCmdState:=999;
		END_IF		
 		
	2://发送启动停止,1011,UINT
		_fbModbusTCP.stParIn.aSendBuffer[1]:=16#00;
		_fbModbusTCP.stParIn.aSendBuffer[2]:=16#00;	
		_fbModbusTCP.stParIn.iHoldingRegisterAddress:=stModbusAddress.iStartStop_Address;
		_fbModbusTCP.stParIn.iHoldingRegisterNum:=1;		 	
		_fbModbusTCP.stOpera.xSetSingalHoldingRegister:=TRUE;
		IF _fbModbusTCP.xDone THEN
			_fbModbusTCP.xExecute:=FALSE;
			_diCmdState:=_diCmdState+1;
		END_IF
		IF _fbModbusTCP.xError THEN
			eERRORID:=RudongPump_ERROR.FLT_Mobdus;
			_diCmdState:=999;
		END_IF	
 		
	3://发送启动停止,2003,UINT
		_fbModbusTCP.stParIn.aSendBuffer[1]:=16#00;
		_fbModbusTCP.stParIn.aSendBuffer[2]:=16#00;	
		_fbModbusTCP.stParIn.iHoldingRegisterAddress:=stModbusAddress.iModuleStartStop_Address;
		_fbModbusTCP.stParIn.iHoldingRegisterNum:=1;		 	
		_fbModbusTCP.stOpera.xSetSingalHoldingRegister:=TRUE;
		IF _fbModbusTCP.xDone THEN
			_fbModbusTCP.xExecute:=FALSE;
			_diCmdState:=_diCmdState+1;
		END_IF
		IF _fbModbusTCP.xError THEN
			eERRORID:=RudongPump_ERROR.FLT_Mobdus;
			_diCmdState:=999;
		END_IF	

	4://完成	
		xComplete:=TRUE;
		
	ELSE
		;
END_CASE
END_METHOD

METHOD PROTECTED ResetAction
VAR_OUTPUT
	xComplete: BOOL;
END_VAR
(*
* Cleaning
* => free all allocated resources
* => reinitialize instance variables
*)
tOperationTimer(IN:=0);
tInvocationTimer(IN:=0);
xRunning:=FALSE;
// init command state
//xExecute:=FALSE;
_diCmdState := 0;
_tonCmdTimeout(in:=FALSE);
_tonDelay(IN:= FALSE);
_tonTimeout(in:=FALSE);
_xModeChange := FALSE;
_rStopCmdTrig(CLK:=FALSE);
_iNGCount := 0;
_fbModbusTCP.xExecute:=FALSE;
FOR k:=1 TO 15 BY 1 DO
	_rOperaTrig[k](CLK:=FALSE);
END_FOR	
	
stDeviceOpe.xConfigure_Auto:= stDeviceOpe.xConfigure_Hmi:= FALSE;
stDeviceOpe.xStop_Auto:= stDeviceOpe.xStop_Hmi:= FALSE;
stDeviceOpe.xFullSpeedPull_Auto:= stDeviceOpe.xFullSpeedPull_Hmi:= FALSE;
stDeviceOpe.xFullSpeedPush_Auto:= stDeviceOpe.xFullSpeedPush_Hmi:= FALSE;
stDeviceOpe.xFullSpeedStop_Auto:= stDeviceOpe.xFullSpeedStop_Hmi:= FALSE;
FOR k:=1 TO 5 DO
	stDeviceOpe.xPull_Auto[k]:= stDeviceOpe.xPull_Hmi[k] := FALSE;
	stDeviceOpe.xPush_Auto[k]:= stDeviceOpe.xPush_Hmi[k] := FALSE;
END_FOR

stDeviceOpe.xPumpCal_Auto:=stDeviceOpe.xPumpCal_Hmi:=FALSE;
stDeviceOpe.xCalParWrite_Auto:=stDeviceOpe.xCalParWrite_Hmi:=FALSE;
stDeviceOpe.xResetCalcoeffCal_Hmi:=FALSE;
xResetRequest:=FALSE;
//复位完成
xComplete:=1;
END_METHOD

END_FUNCTION_BLOCK

// ---- POUs/003_FB/53_RudongPump/41 Modbus指令/FB_ModbusTCP.TcPOU
FUNCTION_BLOCK FB_ModbusTCP
VAR_INPUT
	///参数输入	
	stParIn: ModbusParIn;
	///系统参数输入
	stSysPar: Modbus_SysPar;
	///复位操作
	xResetRequest: BOOL;
	///操作
	stOpera: Modbus_Operation;
	///指令执行
	{attribute 'hide' := ''}
	xExecute: BOOL;
END_VAR
VAR_OUTPUT
	///完成条件满足
	xDone: BOOL;
	///动作正在执行
	xBusy: BOOL;
	///错误条件满足
	xError: BOOL;
	eERRORID: Modbus_ErrorCode;
	eTCPErrorID: UDINT;
	///MODBUS错误码
	sModbusError: STRING;
	///指令被打断，一般是处于急停中
	xAborted: BOOL;
	///代表指令准备完成
	xRdyCmd: BOOL;
	///用于显示的错误代码
	sError: STRING;
	///参数输出
	stParOut: ModbusParOut;
END_VAR
VAR
	///MODBUS TCP收发序列号
	{attribute 'hide' := ''}
	iModbusTCP_ComID: WORD;
	///指令中断
	{attribute 'hide' := ''}
	xAbort: BOOL;
	///接收缓存区域(byte数组)
	{attribute 'hide' := ''}
	_rxBuffer: ARRAY[1..MAX_PLCPRJ_RXBUFFER_SIZE] OF BYTE;
	///执行指令
	{attribute 'hide' := ''}
	eCmd: Modbus_Cmd;
	{attribute 'hide' := ''}
	i: INT;
	{attribute 'hide' := ''}
	j: INT;
	{attribute 'hide' := ''}
	k: INT;
	{attribute 'hide' := ''}
	xOpe: BOOL;
	{attribute 'hide' := ''}
	_diCmdState: DINT;
	{attribute 'hide' := ''}
	_diReadParStep: DINT;
	{attribute 'hide' := ''}
	_fbTcpIpClient: FB_TcpIpClient;
	///当前状态
	{attribute 'hide' := ''}
	eState: STATE;
	{attribute 'hide' := ''}
	xFirstInvocation: BOOL := TRUE;
	{attribute 'hide' := ''}
	xTimeOut: BOOL;
	{attribute 'hide' := ''}
	tOperationTimer: TON;
	{attribute 'hide' := ''}
	_tDelay: TON;
	{attribute 'hide' := ''}
	_twaitDelay: TON;
	{attribute 'hide' := ''}
	_first: BOOL;
	///发送NG计数	
	{attribute 'hide' := ''}
	_iSendNGCount: INT;
	{attribute 'hide' := ''}
	_tonCmdTimeout: TON;
	{attribute 'hide' := ''}
	_tonDelay: TON;
	{attribute 'hide' := ''}
	_tonTimeout: TON;
	{attribute 'hide' := ''}
	_xDone: BOOL;
END_VAR
VAR_TEMP
	xAgain: BOOL;
END_VAR

IF NOT _first 
THEN
	_first := TRUE;
ELSE
	_fbTcpIpClient.nRemotePort := stSysPar.nRemotePort;
	_fbTcpIpClient.sRemoteHost := stSysPar.sRemoteHost;
	xAgain:=0;
	_fbTcpIpClient();
	eTCPErrorID := _fbTcpIpClient.udiErrorID;
	xRdyCmd := ( eState = STATE.DORMANT );
	xDone := _xDone AND xExecute;//判断是否处于当前流程的Done状态
	REPEAT
		CASE eState OF
			STATE.DORMANT:
				HandleDormantState(xAgain=> xAgain);
			STATE.EXECUTING:
				HandleExecutingState(xAgain=> xAgain);
			STATE.DONE:
				HandleDoneState(xAgain=> xAgain);
			STATE.INERROR:
				HandleErrorState(xAgain=> xAgain);
			STATE.ABORTING:
				HandleAbortingState(xAgain=> xAgain);
			STATE.ABORTED:
				HandleAbortedState(xAgain=> xAgain);
			STATE.RESETING:
				HandleResettingState(xAgain=> xAgain);
			END_CASE
	UNTIL (xAgain=0)
	END_REPEAT
END_IF


xOpe:=
stOpera.xReadCoilStatus OR 
stOpera.xReadHoldingRegisters OR 
stOpera.xReadInputRegisters OR 
stOpera.xReadInputStatus OR 
stOpera.xSetMultiCoil OR 
stOpera.xSetMultiHoldingRegister OR 
stOpera.xSetSingalCoil OR 
stOpera.xSetSingalHoldingRegister;

//错误码
CASE eERRORID OF
	Modbus_ErrorCode.FLT_CMD						:	sError:='FLT_CMD';
	Modbus_ErrorCode.FLT_CMDTIMEOUT			:	sError:='FLT_CMDTIMEOUT';
	Modbus_ErrorCode.FLT_MODBUS_ERROR		:	sError:=sModbusError;
	Modbus_ErrorCode.FLT_NoResponse			:	sError:='FLT_NoResponse';
	Modbus_ErrorCode.FLT_PAROVERFLOW		:	sError:='FLT_PAROVERFLOW';	
	Modbus_ErrorCode.FLT_RECEIVE_ERROR	:	sError:='FLT_RECEIVE_ERROR';	
	Modbus_ErrorCode.FLT_SEND_ERROR			:	sError:='FLT_SEND_ERROR';	
	Modbus_ErrorCode.No_ERROR						:	sError:='No_ERROR';	
END_CASE

{attribute 'hide' := ''}
METHOD PROTECTED AbortAction
VAR_OUTPUT
	xComplete: BOOL;
END_VAR
(*
* Cleaning
* => abort all running operation
* => if an NBS.ERROR codition is reached, set eErrorID to a Value rather then NBS.ERROR.NO_ERROR 
*)
xComplete:=1;
eErrorID:=Modbus_ErrorCode.NO_ERROR;
END_METHOD

METHOD Cmd_ReadCoil
VAR_OUTPUT
	xComplete: BOOL;
END_VAR
IF eERRORID <> Modbus_ErrorCode.No_ERROR
THEN
  RETURN;  
END_IF

CASE _diCmdState OF	
	0://清空数据
		_fbTcpIpClient.xEnable := FALSE;	
		_tonDelay(IN:= TRUE,pt:=T#1MS);
		_tonTimeout(IN:= FALSE);
		SysMemSet( ADR(_fbTcpIpClient.aToServer ), 0, SIZEOF(_fbTcpIpClient.aToServer) );//清除发送区域
		SysMemSet( ADR(_rxBuffer ), 0, SIZEOF(_rxBuffer) );//清除接收报告数据缓存区域
		SysMemSet( ADR(stParOut.aRcvBuffer ), 0, SIZEOF(stParOut.aRcvBuffer) );//清除接收报告数据缓存区域		
		SysMemSet( ADR(stParOut.aRcvCoilBuffer ), 0, SIZEOF(stParOut.aRcvCoilBuffer) );//清除接收报告数据缓存区域		
		_fbTcpIpClient.xNeedReceive := TRUE;//默认都是需要有收发交互的	
		_fbTcpIpClient.xNeedDisConnect := TRUE;//默认都是需要有收发交互的		
		IF _tonDelay.Q THEN
			_tonDelay(IN:= FALSE,pt:=T#20MS);
			_diCmdState:=_diCmdState+1;	
		END_IF	
	
	1://拼接指令
		_fbTcpIpClient.aToServer[1] :=TO_BYTE(SHR(iModbusTCP_ComID,8));
		_fbTcpIpClient.aToServer[2] :=TO_BYTE(iModbusTCP_ComID);
		_fbTcpIpClient.aToServer[3] :=16#00;//		
		_fbTcpIpClient.aToServer[4] :=16#00;//
		_fbTcpIpClient.aToServer[5] :=16#00;//		
		_fbTcpIpClient.aToServer[6] :=16#06;//后面发送字节数量,6个字节			
		_fbTcpIpClient.aToServer[7] :=stSysPar.xSlaveAdr;//设备地址
		_fbTcpIpClient.aToServer[8] :=16#01;//查询功能码01
		_fbTcpIpClient.aToServer[9] :=TO_BYTE(SHR(stParIn.iHoldingRegisterAddress,8));
		_fbTcpIpClient.aToServer[10] :=TO_BYTE(stParIn.iHoldingRegisterAddress);      //读取寄存器起始地址 
		_fbTcpIpClient.aToServer[11] :=TO_BYTE(SHR(stParIn.iCoilNum,8));
		_fbTcpIpClient.aToServer[12] :=TO_BYTE(stParIn.iCoilNum);       		//读取寄存器数量
		_fbTcpIpClient.udiSendNumber:=12;
		IF stParIn.iCoilNum>2000 OR stParIn.iCoilNum<1 THEN
			eERRORID:=Modbus_ErrorCode.FLT_PAROVERFLOW	;//参数超出范围
			_diCmdState := 999;			
		END_IF		
		IF _fbTcpIpClient.xRdyCmd
		THEN
			_diCmdState:=_diCmdState+1;
		ELSE
			_fbTcpIpClient.xEnable := FALSE;
		END_IF
		
	2://接收数据
		_fbTcpIpClient.xEnable 		:= TRUE;	
		IF _fbTcpIpClient.xDone//接收成功
		THEN	
			_iSendNgCount 					:= 0;//代表数据接收成功									
			_rxBuffer 							:= _fbTcpIpClient.rxBuffer;							
			_diCmdState:=_diCmdState+1;			
		END_IF
		//发送出错
		IF _fbTcpIpClient.xError 
		THEN//以太网功能报警，一般就是网络建立有问题，此时一般需要去查网络问题
			_iSendNgCount := _iSendNgCount + 1;
			IF _iSendNgCount <= 3//3次重发
			THEN		
				_tDelay(in:=TRUE,PT:=T#100MS);	
				IF _tDelay.Q
				THEN
					_tDelay(in:=FALSE);
					_diCmdState:=0;//重发
				END_IF							
			ELSE			
				eERRORID:=Modbus_ErrorCode.FLT_SEND_ERROR	;//指令发送出错，可能是通信异常	
				_diCmdState := 999;
			END_IF						
		END_IF			
		
	3://校验MODBUS返回指令
		_tonTimeout(IN:= TRUE,pt:=T#3S);
		IF _tonTimeout.Q THEN
			_tonTimeout(IN:=FALSE);
			eERRORID:=Modbus_ErrorCode.FLT_NoResponse	;//无响应
			_diCmdState := 999;			
		END_IF			
		
	//指令返回OK
		IF 
			_rxBuffer[1]=_fbTcpIpClient.aToServer[1] AND
			_rxBuffer[2]=_fbTcpIpClient.aToServer[2] AND
			_rxBuffer[3]=_fbTcpIpClient.aToServer[3] AND
			_rxBuffer[4]=_fbTcpIpClient.aToServer[4] AND
			_rxBuffer[7]=stSysPar.xSlaveAdr AND
			_rxBuffer[8]=16#01//功能码
		THEN
			IF //如果是8的倍数
				stParIn.iCoilNum MOD 8 =0 AND
				_rxBuffer[5]=TO_BYTE(SHR(stParIn.iCoilNum/8+3,8)) AND
				_rxBuffer[6]=TO_BYTE(stParIn.iCoilNum/8+3) AND
				_rxBuffer[9]=TO_BYTE(stParIn.iCoilNum/8)
			THEN
				_diCmdState:=_diCmdState+1;				
			END_IF	
			IF //如果不是8的倍数
				stParIn.iCoilNum MOD 8 <>0 AND
				_rxBuffer[5]=TO_BYTE(SHR(stParIn.iCoilNum/8+4,8)) AND
				_rxBuffer[6]=TO_BYTE(stParIn.iCoilNum/8+4) AND
				_rxBuffer[9]=TO_BYTE(stParIn.iCoilNum/8+1) 
			THEN
				_diCmdState:=_diCmdState+1;				
			END_IF			
		END_IF
		
		//指令返回MODBUS错误码
		IF 
			_rxBuffer[1]=_fbTcpIpClient.aToServer[1] AND
			_rxBuffer[2]=_fbTcpIpClient.aToServer[2] AND
			_rxBuffer[3]=_fbTcpIpClient.aToServer[3] AND
			_rxBuffer[4]=_fbTcpIpClient.aToServer[4] AND
			_rxBuffer[5]=0 AND 
			_rxBuffer[6]=3 AND
			_rxBuffer[7]=_fbTcpIpClient.aToServer[7] AND
			_rxBuffer[8]=16#81//功能码
		THEN
			sModbusError:=ModbusTCP_ErrorQuery(_rxBuffer[9]);//解析MODBUS错误代码
			eERRORID:=Modbus_ErrorCode.FLT_MODBUS_ERROR	;//Modbus错误
			_diCmdState := 999;				
		END_IF		
		
		//指令返回异常,重发3次
		IF 
			_rxBuffer[1]<>_fbTcpIpClient.aToServer[1] OR
			_rxBuffer[2]<>_fbTcpIpClient.aToServer[2] OR
			_rxBuffer[3]<>0 OR
			_rxBuffer[4]<>0 OR
			_rxBuffer[7]<>_fbTcpIpClient.aToServer[7]
		THEN		
			_iSendNgCount := _iSendNgCount + 1;
			IF _iSendNgCount <= 3//3次重发
			THEN		
				_tDelay(in:=TRUE,PT:=T#100MS);	
				IF _tDelay.Q
				THEN
					_tDelay(in:=FALSE);
					_diCmdState:=0;//重发
				END_IF							
			ELSE	
				eERRORID:=Modbus_ErrorCode.FLT_RECEIVE_ERROR	;//接收指令错误
				_diCmdState := 999;
			END_IF		
		END_IF
		
	4://解析数据
		SysMemCpy(ADR(stparout.aRcvBuffer),ADR(_rxBuffer[10]),TO_INT(_rxBuffer[9]));
		iModbusTCP_ComID:=iModbusTCP_ComID+1;
		_diCmdState:=_diCmdState+1;	
		
	5://获取BOOL数据
		FOR i:=1 TO _rxBuffer[9] BY 1 DO		
			stparout.aRcvCoilBuffer[(i-1)*8+1]	:=stparout.aRcvBuffer[i].00;
			stparout.aRcvCoilBuffer[(i-1)*8+2]	:=stparout.aRcvBuffer[i].01;		
			stparout.aRcvCoilBuffer[(i-1)*8+3]	:=stparout.aRcvBuffer[i].02;
			stparout.aRcvCoilBuffer[(i-1)*8+4]	:=stparout.aRcvBuffer[i].03;
			stparout.aRcvCoilBuffer[(i-1)*8+5]	:=stparout.aRcvBuffer[i].04;
			stparout.aRcvCoilBuffer[(i-1)*8+6]	:=stparout.aRcvBuffer[i].05;
			stparout.aRcvCoilBuffer[(i-1)*8+7]	:=stparout.aRcvBuffer[i].06;
			stparout.aRcvCoilBuffer[(i-1)*8+8]	:=stparout.aRcvBuffer[i].07;
		END_FOR
		xComplete:=TRUE;

END_CASE
END_METHOD

METHOD Cmd_ReadHoldingRegister
VAR_OUTPUT
	xComplete: BOOL;
END_VAR
IF eERRORID <> Modbus_ErrorCode.No_ERROR
THEN
  RETURN;  
END_IF

CASE _diCmdState OF	
	0://清空数据
		_fbTcpIpClient.xEnable := FALSE;	
		_tonDelay(IN:= TRUE,pt:=T#1MS);
		_tonTimeout(IN:= FALSE);
		SysMemSet( ADR(_fbTcpIpClient.aToServer ), 0, SIZEOF(_fbTcpIpClient.aToServer) );//清除发送区域
		SysMemSet( ADR(_rxBuffer ), 0, SIZEOF(_rxBuffer) );//清除接收报告数据缓存区域
		SysMemSet( ADR(stParOut.aRcvBuffer ), 0, SIZEOF(stParOut.aRcvBuffer) );//清除接收报告数据缓存区域		
		SysMemSet( ADR(stParOut.aRcvCoilBuffer ), 0, SIZEOF(stParOut.aRcvCoilBuffer) );//清除接收报告数据缓存区域		
		_fbTcpIpClient.xNeedReceive := TRUE;//默认都是需要有收发交互的	
		_fbTcpIpClient.xNeedDisConnect := TRUE;//默认都是需要有收发交互的		
		IF _tonDelay.Q THEN
			_tonDelay(IN:= FALSE,pt:=T#20MS);
			_diCmdState:=_diCmdState+1;	
		END_IF	
	
	1://拼接指令
		_fbTcpIpClient.aToServer[1] :=TO_BYTE(SHR(iModbusTCP_ComID,8));
		_fbTcpIpClient.aToServer[2] :=TO_BYTE(iModbusTCP_ComID);
		_fbTcpIpClient.aToServer[3] :=16#00;//		
		_fbTcpIpClient.aToServer[4] :=16#00;//
		_fbTcpIpClient.aToServer[5] :=16#00;//		
		_fbTcpIpClient.aToServer[6] :=16#06;//后面发送字节数量,6个字节			
		_fbTcpIpClient.aToServer[7] :=stSysPar.xSlaveAdr;//设备地址
		_fbTcpIpClient.aToServer[8] :=16#03;//查询功能码03
		_fbTcpIpClient.aToServer[9] :=TO_BYTE(SHR(stParIn.iHoldingRegisterAddress,8));
		_fbTcpIpClient.aToServer[10] :=TO_BYTE(stParIn.iHoldingRegisterAddress);      //读取寄存器起始地址 
		_fbTcpIpClient.aToServer[11] :=TO_BYTE(SHR(stParIn.iHoldingRegisterNum,8));
		_fbTcpIpClient.aToServer[12] :=TO_BYTE(stParIn.iHoldingRegisterNum);       		//读取寄存器数量
		_fbTcpIpClient.udiSendNumber:=12;
		IF stParIn.iHoldingRegisterNum>125 OR stParIn.iHoldingRegisterNum<1 THEN
			eERRORID:=Modbus_ErrorCode.FLT_PAROVERFLOW	;//参数超出范围
			_diCmdState := 999;			
		END_IF		
		IF _fbTcpIpClient.xRdyCmd
		THEN
			_diCmdState:=_diCmdState+1;
		ELSE
			_fbTcpIpClient.xEnable := FALSE;
		END_IF
		
	2://接收数据
		_fbTcpIpClient.xEnable 		:= TRUE;	
		IF _fbTcpIpClient.xDone//接收成功
		THEN	
			_iSendNgCount 					:= 0;//代表数据接收成功									
			_rxBuffer 							:= _fbTcpIpClient.rxBuffer;							
			_diCmdState:=_diCmdState+1;		
		END_IF
		//发送出错
		IF _fbTcpIpClient.xError 
		THEN//以太网功能报警，一般就是网络建立有问题，此时一般需要去查网络问题
			_iSendNgCount := _iSendNgCount + 1;
			IF _iSendNgCount <= 3//3次重发
			THEN		
				_tDelay(in:=TRUE,PT:=T#100MS);	
				IF _tDelay.Q
				THEN
					_tDelay(in:=FALSE);
					_diCmdState:=0;//重发
				END_IF							
			ELSE			
				eERRORID:=Modbus_ErrorCode.FLT_SEND_ERROR	;//指令发送出错，可能是通信异常	
				_diCmdState := 999;
			END_IF						
		END_IF			
		
	3://校验MODBUS返回指令
		_tonTimeout(IN:= TRUE,pt:=T#3S);
		IF _tonTimeout.Q THEN
			_tonTimeout(IN:=FALSE);
			eERRORID:=Modbus_ErrorCode.FLT_NoResponse	;//无响应
			_diCmdState := 999;			
		END_IF	
		
	//指令返回OK
		IF 
			_rxBuffer[1]=_fbTcpIpClient.aToServer[1] AND
			_rxBuffer[2]=_fbTcpIpClient.aToServer[2] AND
			_rxBuffer[3]=_fbTcpIpClient.aToServer[3] AND
			_rxBuffer[4]=_fbTcpIpClient.aToServer[4] AND
			_rxBuffer[5]=TO_BYTE(SHR((stParIn.iHoldingRegisterNum*2+3),8)) AND //数量
			_rxBuffer[6]=TO_BYTE(stParIn.iHoldingRegisterNum*2+3) AND
			_rxBuffer[7]=stSysPar.xSlaveAdr AND
			_rxBuffer[8]=16#03 AND//功能码
			_rxBuffer[9]=TO_BYTE(stParIn.iHoldingRegisterNum*2)//一次最多读取255个字节,即125个字
		THEN
			_diCmdState:=_diCmdState+1;
		END_IF
		
		//指令返回MODBUS错误码
		IF 
			_rxBuffer[1]=_fbTcpIpClient.aToServer[1] AND
			_rxBuffer[2]=_fbTcpIpClient.aToServer[2] AND
			_rxBuffer[3]=_fbTcpIpClient.aToServer[3] AND
			_rxBuffer[4]=_fbTcpIpClient.aToServer[4] AND
			_rxBuffer[5]=0 AND 
			_rxBuffer[6]=3 AND
			_rxBuffer[7]=_fbTcpIpClient.aToServer[7] AND
			_rxBuffer[8]=16#83//功能码
		THEN
			sModbusError:=ModbusTCP_ErrorQuery(_rxBuffer[9]);//解析MODBUS错误代码
			eERRORID:=Modbus_ErrorCode.FLT_MODBUS_ERROR	;//Modbus错误
			_diCmdState := 999;				
		END_IF		
		
		//指令返回异常,重发3次
		IF 
			_rxBuffer[1]<>_fbTcpIpClient.aToServer[1] OR
			_rxBuffer[2]<>_fbTcpIpClient.aToServer[2] OR
			_rxBuffer[3]<>0 OR
			_rxBuffer[4]<>0 OR
			_rxBuffer[7]<>_fbTcpIpClient.aToServer[7]
		THEN		
			_iSendNgCount := _iSendNgCount + 1;
			IF _iSendNgCount <= 3//3次重发
			THEN		
				_tDelay(in:=TRUE,PT:=T#100MS);	
				IF _tDelay.Q
				THEN
					_tDelay(in:=FALSE);
					_diCmdState:=0;//重发
				END_IF							
			ELSE	
				eERRORID:=Modbus_ErrorCode.FLT_RECEIVE_ERROR	;//接收指令错误
				_diCmdState := 999;
			END_IF		
		END_IF
		
	4://解析数据
		SysMemCpy(ADR(stparout.aRcvBuffer),ADR(_rxBuffer[10]),TO_INT(_rxBuffer[9]));
		iModbusTCP_ComID:=iModbusTCP_ComID+1;
		xComplete:=TRUE;


END_CASE
END_METHOD

METHOD Cmd_ReadInputCoil
VAR_OUTPUT
	xComplete: BOOL;
END_VAR
IF eERRORID <> Modbus_ErrorCode.No_ERROR
THEN
  RETURN;  
END_IF

CASE _diCmdState OF	
	0://清空数据
		_fbTcpIpClient.xEnable := FALSE;	
		_tonDelay(IN:= TRUE,pt:=T#1MS);
		_tonTimeout(IN:= FALSE);
		SysMemSet( ADR(_fbTcpIpClient.aToServer ), 0, SIZEOF(_fbTcpIpClient.aToServer) );//清除发送区域
		SysMemSet( ADR(_rxBuffer ), 0, SIZEOF(_rxBuffer) );//清除接收报告数据缓存区域
		SysMemSet( ADR(stParOut.aRcvBuffer ), 0, SIZEOF(stParOut.aRcvBuffer) );//清除接收报告数据缓存区域	
		SysMemSet( ADR(stParOut.aRcvCoilBuffer ), 0, SIZEOF(stParOut.aRcvCoilBuffer) );//清除接收报告数据缓存区域		
		_fbTcpIpClient.xNeedReceive := TRUE;//默认都是需要有收发交互的	
		_fbTcpIpClient.xNeedDisConnect := TRUE;//默认都是需要有收发交互的		
		IF _tonDelay.Q THEN
			_tonDelay(IN:= FALSE,pt:=T#20MS);
			_diCmdState:=_diCmdState+1;	
		END_IF	
	
	1://拼接指令
		_fbTcpIpClient.aToServer[1] :=TO_BYTE(SHR(iModbusTCP_ComID,8));
		_fbTcpIpClient.aToServer[2] :=TO_BYTE(iModbusTCP_ComID);
		_fbTcpIpClient.aToServer[3] :=16#00;//		
		_fbTcpIpClient.aToServer[4] :=16#00;//
		_fbTcpIpClient.aToServer[5] :=16#00;//		
		_fbTcpIpClient.aToServer[6] :=16#06;//后面发送字节数量,6个字节			
		_fbTcpIpClient.aToServer[7] :=stSysPar.xSlaveAdr;//设备地址
		_fbTcpIpClient.aToServer[8] :=16#02;//查询功能码02
		_fbTcpIpClient.aToServer[9] :=TO_BYTE(SHR(stParIn.iHoldingRegisterAddress,8));
		_fbTcpIpClient.aToServer[10] :=TO_BYTE(stParIn.iHoldingRegisterAddress);      //读取寄存器起始地址 
		_fbTcpIpClient.aToServer[11] :=TO_BYTE(SHR(stParIn.iCoilNum,8));
		_fbTcpIpClient.aToServer[12] :=TO_BYTE(stParIn.iCoilNum);       		//读取寄存器数量
		_fbTcpIpClient.udiSendNumber:=12;
		IF stParIn.iCoilNum>2000 OR stParIn.iCoilNum<1 THEN
			eERRORID:=Modbus_ErrorCode.FLT_PAROVERFLOW	;//参数超出范围
			_diCmdState := 999;			
		END_IF		
		IF _fbTcpIpClient.xRdyCmd
		THEN
			_diCmdState:=_diCmdState+1;
		ELSE
			_fbTcpIpClient.xEnable := FALSE;
		END_IF
		
	2://接收数据
		_fbTcpIpClient.xEnable 		:= TRUE;	
		IF _fbTcpIpClient.xDone//接收成功
		THEN	
			_iSendNgCount 					:= 0;//代表数据接收成功									
			_rxBuffer 							:= _fbTcpIpClient.rxBuffer;							
			_diCmdState:=_diCmdState+1;			
		END_IF
		//发送出错
		IF _fbTcpIpClient.xError 
		THEN//以太网功能报警，一般就是网络建立有问题，此时一般需要去查网络问题
			_iSendNgCount := _iSendNgCount + 1;
			IF _iSendNgCount <= 3//3次重发
			THEN		
				_tDelay(in:=TRUE,PT:=T#100MS);	
				IF _tDelay.Q
				THEN
					_tDelay(in:=FALSE);
					_diCmdState:=0;//重发
				END_IF							
			ELSE			
				eERRORID:=Modbus_ErrorCode.FLT_SEND_ERROR	;//指令发送出错，可能是通信异常	
				_diCmdState := 999;
			END_IF						
		END_IF			
		
	3://校验MODBUS返回指令
		_tonTimeout(IN:= TRUE,pt:=T#3S);
		IF _tonTimeout.Q THEN
			_tonTimeout(IN:=FALSE);
			eERRORID:=Modbus_ErrorCode.FLT_NoResponse	;//无响应
			_diCmdState := 999;			
		END_IF	
		
	//指令返回OK
		IF 
			_rxBuffer[1]=_fbTcpIpClient.aToServer[1] AND
			_rxBuffer[2]=_fbTcpIpClient.aToServer[2] AND
			_rxBuffer[3]=_fbTcpIpClient.aToServer[3] AND
			_rxBuffer[4]=_fbTcpIpClient.aToServer[4] AND
			_rxBuffer[7]=stSysPar.xSlaveAdr AND
			_rxBuffer[8]=16#02//功能码
		THEN
			IF //如果是8的倍数
				stParIn.iCoilNum MOD 8 =0 AND
				_rxBuffer[5]=TO_BYTE(SHR(stParIn.iCoilNum/8+3,8)) AND
				_rxBuffer[6]=TO_BYTE(stParIn.iCoilNum/8+3) AND
				_rxBuffer[9]=TO_BYTE(stParIn.iCoilNum/8)
			THEN
				_diCmdState:=_diCmdState+1;				
			END_IF	
			IF //如果不是8的倍数
				stParIn.iCoilNum MOD 8 <>0 AND
				_rxBuffer[5]=TO_BYTE(SHR(stParIn.iCoilNum/8+4,8)) AND
				_rxBuffer[6]=TO_BYTE(stParIn.iCoilNum/8+4) AND
				_rxBuffer[9]=TO_BYTE(stParIn.iCoilNum/8+1) 
			THEN
				_diCmdState:=_diCmdState+1;				
			END_IF			
		END_IF
		
		//指令返回MODBUS错误码
		IF 
			_rxBuffer[1]=_fbTcpIpClient.aToServer[1] AND
			_rxBuffer[2]=_fbTcpIpClient.aToServer[2] AND
			_rxBuffer[3]=_fbTcpIpClient.aToServer[3] AND
			_rxBuffer[4]=_fbTcpIpClient.aToServer[4] AND
			_rxBuffer[5]=0 AND 
			_rxBuffer[6]=3 AND
			_rxBuffer[7]=_fbTcpIpClient.aToServer[7] AND
			_rxBuffer[8]=16#82//功能码
		THEN
			sModbusError:=ModbusTCP_ErrorQuery(_rxBuffer[9]);//解析MODBUS错误代码
			eERRORID:=Modbus_ErrorCode.FLT_MODBUS_ERROR	;//Modbus错误
			_diCmdState := 999;				
		END_IF		
		
		//指令返回异常,重发3次
		IF 
			_rxBuffer[1]<>_fbTcpIpClient.aToServer[1] OR
			_rxBuffer[2]<>_fbTcpIpClient.aToServer[2] OR
			_rxBuffer[3]<>0 OR
			_rxBuffer[4]<>0 OR
			_rxBuffer[7]<>_fbTcpIpClient.aToServer[7]
		THEN		
			_iSendNgCount := _iSendNgCount + 1;
			IF _iSendNgCount <= 3//3次重发
			THEN		
				_tDelay(in:=TRUE,PT:=T#100MS);	
				IF _tDelay.Q
				THEN
					_tDelay(in:=FALSE);
					_diCmdState:=0;//重发
				END_IF							
			ELSE	
				eERRORID:=Modbus_ErrorCode.FLT_RECEIVE_ERROR	;//接收指令错误
				_diCmdState := 999;
			END_IF		
		END_IF
		
	4://解析数据
		SysMemCpy(ADR(stparout.aRcvBuffer),ADR(_rxBuffer[10]),TO_INT(_rxBuffer[9]));
		iModbusTCP_ComID:=iModbusTCP_ComID+1;
		_diCmdState:=_diCmdState+1;	
		
	5://获取BOOL数据
		FOR i:=1 TO _rxBuffer[9] BY 1 DO		
			stparout.aRcvCoilBuffer[(i-1)*8+1]	:=stparout.aRcvBuffer[i].00;
			stparout.aRcvCoilBuffer[(i-1)*8+2]	:=stparout.aRcvBuffer[i].01;		
			stparout.aRcvCoilBuffer[(i-1)*8+3]	:=stparout.aRcvBuffer[i].02;
			stparout.aRcvCoilBuffer[(i-1)*8+4]	:=stparout.aRcvBuffer[i].03;
			stparout.aRcvCoilBuffer[(i-1)*8+5]	:=stparout.aRcvBuffer[i].04;
			stparout.aRcvCoilBuffer[(i-1)*8+6]	:=stparout.aRcvBuffer[i].05;
			stparout.aRcvCoilBuffer[(i-1)*8+7]	:=stparout.aRcvBuffer[i].06;
			stparout.aRcvCoilBuffer[(i-1)*8+8]	:=stparout.aRcvBuffer[i].07;
		END_FOR
		xComplete:=TRUE;

END_CASE
END_METHOD

METHOD Cmd_ReadInputRegister
VAR_OUTPUT
	xComplete: BOOL;
END_VAR
IF eERRORID <> Modbus_ErrorCode.No_ERROR
THEN
  RETURN;  
END_IF

CASE _diCmdState OF	
	0://清空数据
		_fbTcpIpClient.xEnable := FALSE;	
		_tonDelay(IN:= TRUE,pt:=T#1MS);
		_tonTimeout(IN:= FALSE);
		SysMemSet( ADR(_fbTcpIpClient.aToServer ), 0, SIZEOF(_fbTcpIpClient.aToServer) );//清除发送区域
		SysMemSet( ADR(_rxBuffer ), 0, SIZEOF(_rxBuffer) );//清除接收报告数据缓存区域
		SysMemSet( ADR(stParOut.aRcvBuffer ), 0, SIZEOF(stParOut.aRcvBuffer) );//清除接收报告数据缓存区域	
		SysMemSet( ADR(stParOut.aRcvCoilBuffer ), 0, SIZEOF(stParOut.aRcvCoilBuffer) );//清除接收报告数据缓存区域		
		_fbTcpIpClient.xNeedReceive := TRUE;//默认都是需要有收发交互的	
		_fbTcpIpClient.xNeedDisConnect := TRUE;//默认都是需要有收发交互的		
		IF _tonDelay.Q THEN
			_tonDelay(IN:= FALSE,pt:=T#20MS);
			_diCmdState:=_diCmdState+1;	
		END_IF	
	
	1://拼接指令
		_fbTcpIpClient.aToServer[1] :=TO_BYTE(SHR(iModbusTCP_ComID,8));
		_fbTcpIpClient.aToServer[2] :=TO_BYTE(iModbusTCP_ComID);
		_fbTcpIpClient.aToServer[3] :=16#00;//		
		_fbTcpIpClient.aToServer[4] :=16#00;//
		_fbTcpIpClient.aToServer[5] :=16#00;//		
		_fbTcpIpClient.aToServer[6] :=16#06;//后面发送字节数量,6个字节			
		_fbTcpIpClient.aToServer[7] :=stSysPar.xSlaveAdr;//设备地址
		_fbTcpIpClient.aToServer[8] :=16#04;//查询功能码04
		_fbTcpIpClient.aToServer[9] :=TO_BYTE(SHR(stParIn.iHoldingRegisterAddress,8));
		_fbTcpIpClient.aToServer[10] :=TO_BYTE(stParIn.iHoldingRegisterAddress);      //读取寄存器起始地址 
		_fbTcpIpClient.aToServer[11] :=TO_BYTE(SHR(stParIn.iHoldingRegisterNum,8));
		_fbTcpIpClient.aToServer[12] :=TO_BYTE(stParIn.iHoldingRegisterNum);       		//读取寄存器数量
		_fbTcpIpClient.udiSendNumber:=12;
		IF stParIn.iHoldingRegisterNum>125 OR stParIn.iHoldingRegisterNum<1 THEN
			eERRORID:=Modbus_ErrorCode.FLT_PAROVERFLOW	;//参数超出范围
			_diCmdState := 999;			
		END_IF		
		IF _fbTcpIpClient.xRdyCmd
		THEN
			_diCmdState:=_diCmdState+1;
		ELSE
			_fbTcpIpClient.xEnable := FALSE;
		END_IF
		
	2://接收数据
		_fbTcpIpClient.xEnable 		:= TRUE;	
		IF _fbTcpIpClient.xDone//接收成功
		THEN	
			_iSendNgCount 					:= 0;//代表数据接收成功									
			_rxBuffer 							:= _fbTcpIpClient.rxBuffer;							
			_diCmdState:=_diCmdState+1;			
		END_IF
		//发送出错
		IF _fbTcpIpClient.xError 
		THEN//以太网功能报警，一般就是网络建立有问题，此时一般需要去查网络问题
			_iSendNgCount := _iSendNgCount + 1;
			IF _iSendNgCount <= 3//3次重发
			THEN		
				_tDelay(in:=TRUE,PT:=T#100MS);	
				IF _tDelay.Q
				THEN
					_tDelay(in:=FALSE);
					_diCmdState:=0;//重发
				END_IF							
			ELSE			
				eERRORID:=Modbus_ErrorCode.FLT_SEND_ERROR	;//指令发送出错，可能是通信异常	
				_diCmdState := 999;
			END_IF						
		END_IF			
		
	3://校验MODBUS返回指令
		_tonTimeout(IN:= TRUE,pt:=T#3S);
		IF _tonTimeout.Q THEN
			_tonTimeout(IN:=FALSE);
			eERRORID:=Modbus_ErrorCode.FLT_NoResponse	;//无响应
			_diCmdState := 999;			
		END_IF	
		
	//指令返回OK
		IF 
			_rxBuffer[1]=_fbTcpIpClient.aToServer[1] AND
			_rxBuffer[2]=_fbTcpIpClient.aToServer[2] AND
			_rxBuffer[3]=_fbTcpIpClient.aToServer[3] AND
			_rxBuffer[4]=_fbTcpIpClient.aToServer[4] AND
			_rxBuffer[5]=TO_BYTE(SHR((stParIn.iHoldingRegisterNum*2+3),8)) AND //数量
			_rxBuffer[6]=TO_BYTE(stParIn.iHoldingRegisterNum*2+3) AND
			_rxBuffer[7]=stSysPar.xSlaveAdr AND
			_rxBuffer[8]=16#04 AND//功能码
			_rxBuffer[9]=TO_BYTE(stParIn.iHoldingRegisterNum*2)//一次最多读取255个字节,即125个字
		THEN
			_diCmdState:=_diCmdState+1;
		END_IF
		
		//指令返回MODBUS错误码
		IF 
			_rxBuffer[1]=_fbTcpIpClient.aToServer[1] AND
			_rxBuffer[2]=_fbTcpIpClient.aToServer[2] AND
			_rxBuffer[3]=_fbTcpIpClient.aToServer[3] AND
			_rxBuffer[4]=_fbTcpIpClient.aToServer[4] AND
			_rxBuffer[5]=0 AND 
			_rxBuffer[6]=3 AND
			_rxBuffer[7]=_fbTcpIpClient.aToServer[7] AND
			_rxBuffer[8]=16#84//功能码
		THEN
			sModbusError:=ModbusTCP_ErrorQuery(_rxBuffer[9]);//解析MODBUS错误代码
			eERRORID:=Modbus_ErrorCode.FLT_MODBUS_ERROR	;//Modbus错误
			_diCmdState := 999;				
		END_IF		
		
		//指令返回异常,重发3次
		IF 
			_rxBuffer[1]<>_fbTcpIpClient.aToServer[1] OR
			_rxBuffer[2]<>_fbTcpIpClient.aToServer[2] OR
			_rxBuffer[3]<>0 OR
			_rxBuffer[4]<>0 OR
			_rxBuffer[7]<>_fbTcpIpClient.aToServer[7]
		THEN		
			_iSendNgCount := _iSendNgCount + 1;
			IF _iSendNgCount <= 3//3次重发
			THEN		
				_tDelay(in:=TRUE,PT:=T#100MS);	
				IF _tDelay.Q
				THEN
					_tDelay(in:=FALSE);
					_diCmdState:=0;//重发
				END_IF							
			ELSE	
				eERRORID:=Modbus_ErrorCode.FLT_RECEIVE_ERROR	;//接收指令错误
				_diCmdState := 999;
			END_IF		
		END_IF
		
	4://解析数据
		SysMemCpy(ADR(stparout.aRcvBuffer),ADR(_rxBuffer[10]),TO_INT(_rxBuffer[9]));
		iModbusTCP_ComID:=iModbusTCP_ComID+1;
		xComplete:=TRUE;


END_CASE
END_METHOD

METHOD Cmd_WriteMultiCoil
VAR_OUTPUT
	xComplete: BOOL;
END_VAR
IF eERRORID <> Modbus_ErrorCode.No_ERROR
THEN
  RETURN;  
END_IF

CASE _diCmdState OF	
	0://清空数据
		_fbTcpIpClient.xEnable := FALSE;	
		_tonDelay(IN:= TRUE,pt:=T#1MS);
		_tonTimeout(IN:= FALSE);
		SysMemSet( ADR(_fbTcpIpClient.aToServer ), 0, SIZEOF(_fbTcpIpClient.aToServer) );//清除发送区域
		SysMemSet( ADR(_rxBuffer ), 0, SIZEOF(_rxBuffer) );//清除接收报告数据缓存区域
		SysMemSet( ADR(stParOut.aRcvBuffer ), 0, SIZEOF(stParOut.aRcvBuffer) );//清除接收报告数据缓存区域	
		SysMemSet( ADR(stParOut.aRcvCoilBuffer ), 0, SIZEOF(stParOut.aRcvCoilBuffer) );//清除接收报告数据缓存区域			
		_fbTcpIpClient.xNeedReceive := TRUE;//默认都是需要有收发交互的	
		_fbTcpIpClient.xNeedDisConnect := TRUE;//默认都是需要有收发交互的		
		IF _tonDelay.Q THEN
			_tonDelay(IN:= FALSE,pt:=T#20MS);
			_diCmdState:=_diCmdState+1;	
		END_IF	
	
	1://拼接指令
(******************************************固定段**********************************************)
		_fbTcpIpClient.aToServer[1] :=TO_BYTE(SHR(iModbusTCP_ComID,8));
		_fbTcpIpClient.aToServer[2] :=TO_BYTE(iModbusTCP_ComID);
		_fbTcpIpClient.aToServer[3] :=16#00;//		
		_fbTcpIpClient.aToServer[4] :=16#00;//	
		_fbTcpIpClient.aToServer[7] :=stSysPar.xSlaveAdr;//设备地址
		_fbTcpIpClient.aToServer[8] :=16#0F;//写入单个寄存器功能码15	
		_fbTcpIpClient.aToServer[9] :=TO_BYTE(SHR((stParIn.iCoilStartAddress),8));//起始地址高位
		_fbTcpIpClient.aToServer[10] :=TO_BYTE(stParIn.iCoilStartAddress); //起始地址低位
		_fbTcpIpClient.aToServer[11] :=TO_BYTE(SHR(stParIn.iCoilNum,8));//写入线圈数量高位
		_fbTcpIpClient.aToServer[12] :=TO_BYTE(stParIn.iCoilNum);//写入线圈数量低位
(******************************************可变段**********************************************)
		IF stParIn.iCoilNum MOD 8 <>0 THEN	
			_fbTcpIpClient.aToServer[13] :=TO_BYTE(stParIn.iCoilNum/8+1);	//写入字节数量
		ELSE
			_fbTcpIpClient.aToServer[13] :=TO_BYTE(stParIn.iCoilNum/8);	//写入字节数量
		END_IF
		_fbTcpIpClient.aToServer[5] :=16#00;//		
		_fbTcpIpClient.aToServer[6] :=TO_BYTE(_fbTcpIpClient.aToServer[13]+7);//后面发送字节数量	
		FOR i:=1 TO _fbTcpIpClient.aToServer[13] BY 1 DO
				_fbTcpIpClient.aToServer[13+i] :=stParIn.aSendBuffer[i];
		END_FOR
		//发送字节长度
		_fbTcpIpClient.udiSendNumber:=_fbTcpIpClient.aToServer[5]*255+_fbTcpIpClient.aToServer[6]+6;	
		IF _fbTcpIpClient.xRdyCmd
		THEN
			_diCmdState:=_diCmdState+1;
		ELSE
			_fbTcpIpClient.xEnable := FALSE;
		END_IF
		
	2://接收数据
		_fbTcpIpClient.xEnable 		:= TRUE;	
		IF _fbTcpIpClient.xDone//接收成功
		THEN	
			_iSendNgCount 					:= 0;//代表数据接收成功									
			_rxBuffer 							:= _fbTcpIpClient.rxBuffer;							
			_diCmdState:=_diCmdState+1;			
		END_IF
		//发送出错
		IF _fbTcpIpClient.xError 
		THEN//以太网功能报警，一般就是网络建立有问题，此时一般需要去查网络问题
			_iSendNgCount := _iSendNgCount + 1;
			IF _iSendNgCount <= 3//3次重发
			THEN		
				_tDelay(in:=TRUE,PT:=T#100MS);	
				IF _tDelay.Q
				THEN
					_tDelay(in:=FALSE);
					_diCmdState:=0;//重发
				END_IF							
			ELSE			
				eERRORID:=Modbus_ErrorCode.FLT_SEND_ERROR	;//指令发送出错，可能是通信异常	
				_diCmdState := 999;
			END_IF						
		END_IF			
		
	3://校验MODBUS返回指令
		_tonTimeout(IN:= TRUE,pt:=T#3S);
		IF _tonTimeout.Q THEN
			_tonTimeout(IN:=FALSE);
			eERRORID:=Modbus_ErrorCode.FLT_NoResponse	;//无响应
			_diCmdState := 999;			
		END_IF	
		
	//指令返回OK
		IF 
			_rxBuffer[1]=_fbTcpIpClient.aToServer[1] AND
			_rxBuffer[2]=_fbTcpIpClient.aToServer[2] AND
			_rxBuffer[3]=_fbTcpIpClient.aToServer[3] AND
			_rxBuffer[4]=_fbTcpIpClient.aToServer[4] AND
			_rxBuffer[5]=_fbTcpIpClient.aToServer[5] AND
			_rxBuffer[6]=16#06 AND
			_rxBuffer[7]=_fbTcpIpClient.aToServer[7] AND
			_rxBuffer[8]=_fbTcpIpClient.aToServer[8] AND
			_rxBuffer[9]=_fbTcpIpClient.aToServer[9] AND 
			_rxBuffer[10]=_fbTcpIpClient.aToServer[10]AND 	
			_rxBuffer[11]=_fbTcpIpClient.aToServer[11]AND
			_rxBuffer[12]=_fbTcpIpClient.aToServer[12]
		THEN
			_diCmdState:=_diCmdState+1;
		END_IF
		
		//指令返回MODBUS错误码
		IF 
			_rxBuffer[1]=_fbTcpIpClient.aToServer[1] AND
			_rxBuffer[2]=_fbTcpIpClient.aToServer[2] AND
			_rxBuffer[3]=_fbTcpIpClient.aToServer[3] AND
			_rxBuffer[4]=_fbTcpIpClient.aToServer[4] AND
			_rxBuffer[5]=_fbTcpIpClient.aToServer[5] AND 
			_rxBuffer[6]=16#03 AND
			_rxBuffer[7]=_fbTcpIpClient.aToServer[7] AND
			_rxBuffer[8]=16#8F//功能码
		THEN
			sModbusError:=ModbusTCP_ErrorQuery(_rxBuffer[9]);//解析MODBUS错误代码
			eERRORID:=Modbus_ErrorCode.FLT_MODBUS_ERROR	;//Modbus错误
			_diCmdState := 999;				
		END_IF		
		
		//指令返回异常,重发3次
		IF 
			_rxBuffer[1]<>_fbTcpIpClient.aToServer[1] OR
			_rxBuffer[2]<>_fbTcpIpClient.aToServer[2] OR
			_rxBuffer[3]<>_fbTcpIpClient.aToServer[3] OR
			_rxBuffer[4]<>_fbTcpIpClient.aToServer[4] OR
			_rxBuffer[7]<>_fbTcpIpClient.aToServer[7]
		THEN		
			_iSendNgCount := _iSendNgCount + 1;
			IF _iSendNgCount <= 3//3次重发
			THEN		
				_tDelay(in:=TRUE,PT:=T#100MS);	
				IF _tDelay.Q
				THEN
					_tDelay(in:=FALSE);
					_diCmdState:=0;//重发
				END_IF							
			ELSE	
				eERRORID:=Modbus_ErrorCode.FLT_RECEIVE_ERROR	;//接收指令错误
				_diCmdState := 999;
			END_IF		
		END_IF
		
	4://解析数据
		xComplete:=TRUE;


END_CASE
END_METHOD

METHOD Cmd_WriteMultiHoldingRegister
VAR_OUTPUT
	xComplete: BOOL;
END_VAR
IF eERRORID <> Modbus_ErrorCode.No_ERROR
THEN
  RETURN;  
END_IF

CASE _diCmdState OF	
	0://清空数据
		_fbTcpIpClient.xEnable := FALSE;	
		_tonDelay(IN:= TRUE,pt:=T#1MS);
		_tonTimeout(IN:= FALSE);
		SysMemSet( ADR(_fbTcpIpClient.aToServer ), 0, SIZEOF(_fbTcpIpClient.aToServer) );//清除发送区域
		SysMemSet( ADR(_rxBuffer ), 0, SIZEOF(_rxBuffer) );//清除接收报告数据缓存区域
		SysMemSet( ADR(stParOut.aRcvBuffer ), 0, SIZEOF(stParOut.aRcvBuffer) );//清除接收报告数据缓存区域	
		SysMemSet( ADR(stParOut.aRcvCoilBuffer ), 0, SIZEOF(stParOut.aRcvCoilBuffer) );//清除接收报告数据缓存区域			
		_fbTcpIpClient.xNeedReceive := TRUE;//默认都是需要有收发交互的	
		_fbTcpIpClient.xNeedDisConnect := TRUE;//默认都是需要有收发交互的		
		IF _tonDelay.Q THEN
			_tonDelay(IN:= FALSE,pt:=T#20MS);
			_diCmdState:=_diCmdState+1;	
		END_IF	
	
	1://拼接指令
(******************************************固定段**********************************************)
		_fbTcpIpClient.aToServer[1] :=TO_BYTE(SHR(iModbusTCP_ComID,8));
		_fbTcpIpClient.aToServer[2] :=TO_BYTE(iModbusTCP_ComID);
		_fbTcpIpClient.aToServer[3] :=16#00;//		
		_fbTcpIpClient.aToServer[4] :=16#00;//
		_fbTcpIpClient.aToServer[5] :=TO_BYTE(SHR(stParIn.iHoldingRegisterNum*2+7,8));//		
		_fbTcpIpClient.aToServer[6] :=TO_BYTE(stParIn.iHoldingRegisterNum*2+7);//后面发送字节数量		
		_fbTcpIpClient.aToServer[7] :=stSysPar.xSlaveAdr;//设备地址
		_fbTcpIpClient.aToServer[8] :=16#10;//写入单个寄存器功能码16		
		_fbTcpIpClient.aToServer[9] :=TO_BYTE(SHR((stParIn.iHoldingRegisterAddress),8));//起始地址高位
		_fbTcpIpClient.aToServer[10] :=TO_BYTE(stParIn.iHoldingRegisterAddress); //起始地址低位
		_fbTcpIpClient.aToServer[11] :=TO_BYTE(SHR(stParIn.iHoldingRegisterNum,8));//写入寄存器数量高位
		_fbTcpIpClient.aToServer[12] :=TO_BYTE(stParIn.iHoldingRegisterNum);//写入寄存器数量低位
(******************************************可变段**********************************************)
		_fbTcpIpClient.aToServer[13] :=TO_BYTE(stParIn.iHoldingRegisterNum*2);	//写入字节数量
		FOR i:=1 TO stParIn.iHoldingRegisterNum*2 DO
			_fbTcpIpClient.aToServer[13+i] :=stParIn.aSendBuffer[i];
			_fbTcpIpClient.aToServer[14+i] :=stParIn.aSendBuffer[i+1];
		END_FOR
		
		_fbTcpIpClient.udiSendNumber:=13+stParIn.iHoldingRegisterNum*2;	
		IF _fbTcpIpClient.xRdyCmd
		THEN
			_diCmdState:=_diCmdState+1;
		ELSE
			_fbTcpIpClient.xEnable := FALSE;
		END_IF
		
	2://接收数据
		_fbTcpIpClient.xEnable 		:= TRUE;	
		IF _fbTcpIpClient.xDone//接收成功
		THEN	
			_iSendNgCount 					:= 0;//代表数据接收成功									
			_rxBuffer 							:= _fbTcpIpClient.rxBuffer;							
			_diCmdState:=_diCmdState+1;			
		END_IF
		//发送出错
		IF _fbTcpIpClient.xError 
		THEN//以太网功能报警，一般就是网络建立有问题，此时一般需要去查网络问题
			_iSendNgCount := _iSendNgCount + 1;
			IF _iSendNgCount <= 3//3次重发
			THEN		
				_tDelay(in:=TRUE,PT:=T#100MS);	
				IF _tDelay.Q
				THEN
					_tDelay(in:=FALSE);
					_diCmdState:=0;//重发
				END_IF							
			ELSE			
				eERRORID:=Modbus_ErrorCode.FLT_SEND_ERROR	;//指令发送出错，可能是通信异常	
				_diCmdState := 999;
			END_IF						
		END_IF			
		
	3://校验MODBUS返回指令
		_tonTimeout(IN:= TRUE,pt:=T#3S);
		IF _tonTimeout.Q THEN
			_tonTimeout(IN:=FALSE);
			eERRORID:=Modbus_ErrorCode.FLT_NoResponse	;//无响应
			_diCmdState := 999;			
		END_IF	
		
	//指令返回OK
		IF 
			_rxBuffer[1]=_fbTcpIpClient.aToServer[1] AND
			_rxBuffer[2]=_fbTcpIpClient.aToServer[2] AND
			_rxBuffer[3]=_fbTcpIpClient.aToServer[3] AND
			_rxBuffer[4]=_fbTcpIpClient.aToServer[4] AND
			_rxBuffer[5]=_fbTcpIpClient.aToServer[5] AND
			_rxBuffer[6]=16#06 AND
			_rxBuffer[7]=_fbTcpIpClient.aToServer[7] AND
			_rxBuffer[8]=_fbTcpIpClient.aToServer[8] AND
			_rxBuffer[9]=_fbTcpIpClient.aToServer[9] AND 
			_rxBuffer[10]=_fbTcpIpClient.aToServer[10]AND 	
			_rxBuffer[11]=_fbTcpIpClient.aToServer[11]AND
			_rxBuffer[12]=_fbTcpIpClient.aToServer[12]
		THEN
			_diCmdState:=_diCmdState+1;
		END_IF
		
		//指令返回MODBUS错误码
		IF 
			_rxBuffer[1]=_fbTcpIpClient.aToServer[1] AND
			_rxBuffer[2]=_fbTcpIpClient.aToServer[2] AND
			_rxBuffer[3]=_fbTcpIpClient.aToServer[3] AND
			_rxBuffer[4]=_fbTcpIpClient.aToServer[4] AND
			_rxBuffer[5]=_fbTcpIpClient.aToServer[5] AND 
			_rxBuffer[6]=16#03 AND
			_rxBuffer[7]=_fbTcpIpClient.aToServer[7] AND
			_rxBuffer[8]=16#90//功能码
		THEN
			sModbusError:=ModbusTCP_ErrorQuery(_rxBuffer[9]);//解析MODBUS错误代码
			eERRORID:=Modbus_ErrorCode.FLT_MODBUS_ERROR	;//Modbus错误
			_diCmdState := 999;				
		END_IF		
		
		//指令返回异常,重发3次
		IF 
			_rxBuffer[1]<>_fbTcpIpClient.aToServer[1] OR
			_rxBuffer[2]<>_fbTcpIpClient.aToServer[2] OR
			_rxBuffer[3]<>_fbTcpIpClient.aToServer[3] OR
			_rxBuffer[4]<>_fbTcpIpClient.aToServer[4] OR
			_rxBuffer[7]<>_fbTcpIpClient.aToServer[7]
		THEN		
			_iSendNgCount := _iSendNgCount + 1;
			IF _iSendNgCount <= 3//3次重发
			THEN		
				_tDelay(in:=TRUE,PT:=T#100MS);	
				IF _tDelay.Q
				THEN
					_tDelay(in:=FALSE);
					_diCmdState:=0;//重发
				END_IF							
			ELSE	
				eERRORID:=Modbus_ErrorCode.FLT_RECEIVE_ERROR	;//接收指令错误
				_diCmdState := 999;
			END_IF		
		END_IF
		
	4://解析数据
		SysMemCpy(ADR(stparout.aRcvBuffer),ADR(_fbTcpIpClient.aToServer[14]),stParIn.iHoldingRegisterNum*2);
		xComplete:=TRUE;


END_CASE
END_METHOD

METHOD Cmd_WriteSingleCoil
VAR_OUTPUT
	xComplete: BOOL;
END_VAR
IF eERRORID <> Modbus_ErrorCode.No_ERROR
THEN
  RETURN;  
END_IF

CASE _diCmdState OF	
	0://清空数据
		_fbTcpIpClient.xEnable := FALSE;	
		_tonDelay(IN:= TRUE,pt:=T#1MS);
		_tonTimeout(IN:= FALSE);
		SysMemSet( ADR(_fbTcpIpClient.aToServer ), 0, SIZEOF(_fbTcpIpClient.aToServer) );//清除发送区域
		SysMemSet( ADR(_rxBuffer ), 0, SIZEOF(_rxBuffer) );//清除接收报告数据缓存区域
		SysMemSet( ADR(stParOut.aRcvBuffer ), 0, SIZEOF(stParOut.aRcvBuffer) );//清除接收报告数据缓存区域	
		SysMemSet( ADR(stParOut.aRcvCoilBuffer ), 0, SIZEOF(stParOut.aRcvCoilBuffer) );//清除接收报告数据缓存区域			
		_fbTcpIpClient.xNeedReceive := TRUE;//默认都是需要有收发交互的	
		_fbTcpIpClient.xNeedDisConnect := TRUE;//默认都是需要有收发交互的		
		IF _tonDelay.Q THEN
			_tonDelay(IN:= FALSE,pt:=T#20MS);
			_diCmdState:=_diCmdState+1;	
		END_IF	
	
	1://拼接指令
		_fbTcpIpClient.aToServer[1] :=TO_BYTE(SHR(iModbusTCP_ComID,8));
		_fbTcpIpClient.aToServer[2] :=TO_BYTE(iModbusTCP_ComID);
		_fbTcpIpClient.aToServer[3] :=16#00;//		
		_fbTcpIpClient.aToServer[4] :=16#00;//
		_fbTcpIpClient.aToServer[5] :=16#00;//		
		_fbTcpIpClient.aToServer[6] :=16#06;//后面发送字节数量,6个字节			
		_fbTcpIpClient.aToServer[7] :=stSysPar.xSlaveAdr;//设备地址
		_fbTcpIpClient.aToServer[8] :=16#05;//写入单个寄存器功能码06
		_fbTcpIpClient.aToServer[9] :=TO_BYTE(SHR(stParIn.iCoilStartAddress,8));
		_fbTcpIpClient.aToServer[10] :=TO_BYTE(stParIn.iCoilStartAddress);   //起始地址 
		IF stParIn.aSendBuffer[1]<>0 THEN
			_fbTcpIpClient.aToServer[11] :=16#FF;//写入寄存器值,固定格式
		ELSE
			_fbTcpIpClient.aToServer[11] :=16#00;//写入寄存器值,固定格式
		END_IF		
		_fbTcpIpClient.aToServer[12] :=16#00;
		_fbTcpIpClient.udiSendNumber:=12;	
		IF _fbTcpIpClient.xRdyCmd
		THEN
			_diCmdState:=_diCmdState+1;
		ELSE
			_fbTcpIpClient.xEnable := FALSE;
		END_IF
		
	2://接收数据
		_fbTcpIpClient.xEnable 		:= TRUE;	
		IF _fbTcpIpClient.xDone//接收成功
		THEN	
			_iSendNgCount 					:= 0;//代表数据接收成功									
			_rxBuffer 							:= _fbTcpIpClient.rxBuffer;							
			_diCmdState:=_diCmdState+1;			
		END_IF
		//发送出错
		IF _fbTcpIpClient.xError 
		THEN//以太网功能报警，一般就是网络建立有问题，此时一般需要去查网络问题
			_iSendNgCount := _iSendNgCount + 1;
			IF _iSendNgCount <= 3//3次重发
			THEN		
				_tDelay(in:=TRUE,PT:=T#100MS);	
				IF _tDelay.Q
				THEN
					_tDelay(in:=FALSE);
					_diCmdState:=0;//重发
				END_IF							
			ELSE			
				eERRORID:=Modbus_ErrorCode.FLT_SEND_ERROR	;//指令发送出错，可能是通信异常	
				_diCmdState := 999;
			END_IF						
		END_IF			
		
	3://校验MODBUS返回指令
		_tonTimeout(IN:= TRUE,pt:=T#3S);
		IF _tonTimeout.Q THEN
			_tonTimeout(IN:=FALSE);
			eERRORID:=Modbus_ErrorCode.FLT_NoResponse	;//无响应
			_diCmdState := 999;			
		END_IF	
		
	//指令返回OK
		IF 
			_rxBuffer[1]=_fbTcpIpClient.aToServer[1] AND
			_rxBuffer[2]=_fbTcpIpClient.aToServer[2] AND
			_rxBuffer[3]=_fbTcpIpClient.aToServer[3] AND
			_rxBuffer[4]=_fbTcpIpClient.aToServer[4] AND
			_rxBuffer[5]=_fbTcpIpClient.aToServer[5] AND
			_rxBuffer[6]=_fbTcpIpClient.aToServer[6] AND
			_rxBuffer[7]=_fbTcpIpClient.aToServer[7] AND
			_rxBuffer[8]=_fbTcpIpClient.aToServer[8] AND
			_rxBuffer[9]=_fbTcpIpClient.aToServer[9] AND 
			_rxBuffer[10]=_fbTcpIpClient.aToServer[10]AND 	
			_rxBuffer[11]=_fbTcpIpClient.aToServer[11]AND
			_rxBuffer[12]=_fbTcpIpClient.aToServer[12]
		THEN
			_diCmdState:=_diCmdState+1;
		END_IF
		
		//指令返回MODBUS错误码
		IF 
			_rxBuffer[1]=_fbTcpIpClient.aToServer[1] AND
			_rxBuffer[2]=_fbTcpIpClient.aToServer[2] AND
			_rxBuffer[3]=_fbTcpIpClient.aToServer[3] AND
			_rxBuffer[4]=_fbTcpIpClient.aToServer[4] AND
			_rxBuffer[5]=_fbTcpIpClient.aToServer[5] AND 
			_rxBuffer[6]=16#03 AND
			_rxBuffer[7]=_fbTcpIpClient.aToServer[7] AND
			_rxBuffer[8]=16#85//功能码
		THEN
			sModbusError:=ModbusTCP_ErrorQuery(_rxBuffer[9]);//解析MODBUS错误代码
			eERRORID:=Modbus_ErrorCode.FLT_MODBUS_ERROR	;//Modbus错误
			_diCmdState := 999;				
		END_IF		
		
		//指令返回异常,重发3次
		IF 
			_rxBuffer[1]<>_fbTcpIpClient.aToServer[1] OR
			_rxBuffer[2]<>_fbTcpIpClient.aToServer[2] OR
			_rxBuffer[3]<>_fbTcpIpClient.aToServer[3] OR
			_rxBuffer[4]<>_fbTcpIpClient.aToServer[4] OR
			_rxBuffer[7]<>_fbTcpIpClient.aToServer[7]
		THEN		
			_iSendNgCount := _iSendNgCount + 1;
			IF _iSendNgCount <= 3//3次重发
			THEN		
				_tDelay(in:=TRUE,PT:=T#100MS);	
				IF _tDelay.Q
				THEN
					_tDelay(in:=FALSE);
					_diCmdState:=0;//重发
				END_IF							
			ELSE	
				eERRORID:=Modbus_ErrorCode.FLT_RECEIVE_ERROR	;//接收指令错误
				_diCmdState := 999;
			END_IF		
		END_IF
		
	4://解析数据
		iModbusTCP_ComID:=iModbusTCP_ComID+1;
		xComplete:=TRUE;


END_CASE
END_METHOD

METHOD Cmd_WriteSingleHoldingRegister
VAR_OUTPUT
	xComplete: BOOL;
END_VAR
IF eERRORID <> Modbus_ErrorCode.No_ERROR
THEN
  RETURN;  
END_IF

CASE _diCmdState OF	
	0://清空数据
		_fbTcpIpClient.xEnable := FALSE;	
		_tonDelay(IN:= TRUE,pt:=T#1MS);
		_tonTimeout(IN:= FALSE);
		SysMemSet( ADR(_fbTcpIpClient.aToServer ), 0, SIZEOF(_fbTcpIpClient.aToServer) );//清除发送区域
		SysMemSet( ADR(_rxBuffer ), 0, SIZEOF(_rxBuffer) );//清除接收报告数据缓存区域
		SysMemSet( ADR(stParOut.aRcvBuffer ), 0, SIZEOF(stParOut.aRcvBuffer) );//清除接收报告数据缓存区域	
		SysMemSet( ADR(stParOut.aRcvCoilBuffer ), 0, SIZEOF(stParOut.aRcvCoilBuffer) );//清除接收报告数据缓存区域			
		_fbTcpIpClient.xNeedReceive := TRUE;//默认都是需要有收发交互的	
		_fbTcpIpClient.xNeedDisConnect := TRUE;//默认都是需要有收发交互的		
		IF _tonDelay.Q THEN
			_tonDelay(IN:= FALSE,pt:=T#20MS);
			_diCmdState:=_diCmdState+1;	
		END_IF	
	
	1://拼接指令
		_fbTcpIpClient.aToServer[1] :=TO_BYTE(SHR(iModbusTCP_ComID,8));
		_fbTcpIpClient.aToServer[2] :=TO_BYTE(iModbusTCP_ComID);
		_fbTcpIpClient.aToServer[3] :=16#00;//		
		_fbTcpIpClient.aToServer[4] :=16#00;//
		_fbTcpIpClient.aToServer[5] :=16#00;//		
		_fbTcpIpClient.aToServer[6] :=16#06;//后面发送字节数量,6个字节			
		_fbTcpIpClient.aToServer[7] :=stSysPar.xSlaveAdr;//设备地址
		_fbTcpIpClient.aToServer[8] :=16#06;//写入单个寄存器功能码06
		_fbTcpIpClient.aToServer[9] :=TO_BYTE(SHR(stParIn.iHoldingRegisterAddress,8));
		_fbTcpIpClient.aToServer[10] :=TO_BYTE(stParIn.iHoldingRegisterAddress);      //读取寄存器起始地址 
		_fbTcpIpClient.aToServer[11] :=stParIn.aSendBuffer[1];
		_fbTcpIpClient.aToServer[12] :=stParIn.aSendBuffer[2];//写入寄存器值
		_fbTcpIpClient.udiSendNumber:=12;	
		IF _fbTcpIpClient.xRdyCmd
		THEN
			_diCmdState:=_diCmdState+1;
		ELSE
			_fbTcpIpClient.xEnable := FALSE;
		END_IF
		
	2://接收数据
		_fbTcpIpClient.xEnable 		:= TRUE;	
		IF _fbTcpIpClient.xDone//接收成功
		THEN	
			_iSendNgCount 					:= 0;//代表数据接收成功									
			_rxBuffer 							:= _fbTcpIpClient.rxBuffer;							
			_diCmdState:=_diCmdState+1;			
		END_IF
		//发送出错
		IF _fbTcpIpClient.xError 
		THEN//以太网功能报警，一般就是网络建立有问题，此时一般需要去查网络问题
			_iSendNgCount := _iSendNgCount + 1;
			IF _iSendNgCount <= 3//3次重发
			THEN		
				_tDelay(in:=TRUE,PT:=T#100MS);	
				IF _tDelay.Q
				THEN
					_tDelay(in:=FALSE);
					_diCmdState:=0;//重发
				END_IF							
			ELSE			
				eERRORID:=Modbus_ErrorCode.FLT_SEND_ERROR	;//指令发送出错，可能是通信异常	
				_diCmdState := 999;
			END_IF						
		END_IF			
		
	3://校验MODBUS返回指令
		_tonTimeout(IN:= TRUE,pt:=T#3S);
		IF _tonTimeout.Q THEN
			_tonTimeout(IN:=FALSE);
			eERRORID:=Modbus_ErrorCode.FLT_NoResponse	;//无响应
			_diCmdState := 999;			
		END_IF	
		
	//指令返回OK
		IF 
			_rxBuffer[1]=_fbTcpIpClient.aToServer[1] AND
			_rxBuffer[2]=_fbTcpIpClient.aToServer[2] AND
			_rxBuffer[3]=_fbTcpIpClient.aToServer[3] AND
			_rxBuffer[4]=_fbTcpIpClient.aToServer[4] AND
			_rxBuffer[5]=_fbTcpIpClient.aToServer[5] AND
			_rxBuffer[6]=_fbTcpIpClient.aToServer[6] AND
			_rxBuffer[7]=_fbTcpIpClient.aToServer[7] AND
			_rxBuffer[8]=_fbTcpIpClient.aToServer[8] AND
			_rxBuffer[9]=_fbTcpIpClient.aToServer[9] AND 
			_rxBuffer[10]=_fbTcpIpClient.aToServer[10]AND 	
			_rxBuffer[11]=_fbTcpIpClient.aToServer[11]AND
			_rxBuffer[12]=_fbTcpIpClient.aToServer[12]
		THEN
			_diCmdState:=_diCmdState+1;
		END_IF
		
		//指令返回MODBUS错误码
		IF 
			_rxBuffer[1]=_fbTcpIpClient.aToServer[1] AND
			_rxBuffer[2]=_fbTcpIpClient.aToServer[2] AND
			_rxBuffer[3]=_fbTcpIpClient.aToServer[3] AND
			_rxBuffer[4]=_fbTcpIpClient.aToServer[4] AND
			_rxBuffer[5]=_fbTcpIpClient.aToServer[5] AND 
			_rxBuffer[6]=16#03 AND
			_rxBuffer[7]=_fbTcpIpClient.aToServer[7] AND
			_rxBuffer[8]=16#86//功能码
		THEN
			sModbusError:=ModbusTCP_ErrorQuery(_rxBuffer[9]);//解析MODBUS错误代码
			eERRORID:=Modbus_ErrorCode.FLT_MODBUS_ERROR	;//Modbus错误
			_diCmdState := 999;				
		END_IF		
		
		//指令返回异常,重发3次
		IF 
			_rxBuffer[1]<>_fbTcpIpClient.aToServer[1] OR
			_rxBuffer[2]<>_fbTcpIpClient.aToServer[2] OR
			_rxBuffer[3]<>_fbTcpIpClient.aToServer[3] OR
			_rxBuffer[4]<>_fbTcpIpClient.aToServer[4] OR
			_rxBuffer[7]<>_fbTcpIpClient.aToServer[7]
		THEN		
			_iSendNgCount := _iSendNgCount + 1;
			IF _iSendNgCount <= 3//3次重发
			THEN		
				_tDelay(in:=TRUE,PT:=T#100MS);	
				IF _tDelay.Q
				THEN
					_tDelay(in:=FALSE);
					_diCmdState:=0;//重发
				END_IF							
			ELSE	
				eERRORID:=Modbus_ErrorCode.FLT_RECEIVE_ERROR	;//接收指令错误
				_diCmdState := 999;
			END_IF		
		END_IF
		
	4://解析数据
		SysMemCpy(ADR(stparout.aRcvBuffer),ADR(_rxBuffer[11]),2);
		iModbusTCP_ComID:=iModbusTCP_ComID+1;
		xComplete:=TRUE;


END_CASE
END_METHOD

{attribute 'hide' := ''}
METHOD PROTECTED CyclicAction
VAR_OUTPUT
	xComplete: BOOL;
END_VAR
IF xAbort=0 THEN
    IF xFirstInvocation THEN
    (*
    * Staring
    * for then first (!) invocaion,
    * sample then input variables
    *)			
      _diCmdState:= 0;
			_iSendNgCount := 0;
			xFirstInvocation:=0;			
    END_IF  
		REPEAT
			//	
			IF stSysPar.xSlaveAdr=0 THEN
				_fbTcpIpClient.xNeedReceive:=FALSE;//广播模式不需要返回数据
			ELSE
				_fbTcpIpClient.xNeedReceive:=TRUE;//非广播模式需要返回数据
			END_IF


			CASE eCmd OF//判断指令类型
				Modbus_Cmd.ReadCoilStatus://读取线圈,01
						Cmd_ReadCoil(xComplete=> xComplete);	

				Modbus_Cmd.ReadInputStatus://读取线圈,02
						Cmd_ReadInputCoil(xComplete=> xComplete);
			
				Modbus_Cmd.ReadHoldingRegisters://读取保持寄存器,03
						Cmd_ReadHoldingRegister(xComplete=> xComplete);

				Modbus_Cmd.ReadInputRegisters://读取保持寄存器,04
						Cmd_ReadInputRegister(xComplete=> xComplete);
	
				Modbus_Cmd.SetSingalCoil://写入单个线圈,05
						Cmd_WriteSingleCoil(xComplete=> xComplete);	
					
				Modbus_Cmd.SetSingalHoldingRegister://写入单个保持寄存器,06
						Cmd_WriteSingleHoldingRegister(xComplete=> xComplete);

				Modbus_Cmd.SetMultiCoil://写入多个线圈,15
						Cmd_WriteMultiCoil(xComplete=> xComplete);
						
				Modbus_Cmd.SetMultiHoldingRegister://写入多个保持寄存器,16
						Cmd_WriteMultiHoldingRegister(xComplete=> xComplete);
						
				ELSE
					;	
				END_CASE		   
      UNTIL (TRUE)
	END_REPEAT
END_IF

IF xAbort OR xComplete OR eERRORID<>Modbus_ErrorCode.No_ERROR THEN    
    (*
    * Cleaning
    * => free as much allocated resources as possible
    *)    
    tOperationTimer(IN:=0);
END_IF
END_METHOD

{attribute 'hide' := ''}
METHOD PRIVATE FINAL HandleAbortedState
VAR_INPUT
END_VAR
VAR_OUTPUT
	xAgain: BOOL;
END_VAR
VAR
	xComplete: BOOL;
END_VAR
IF xAborted AND xResetRequest THEN
    eState:=STATE.RESETING;
    xAgain:=1;
ELSE
    xBusy:=0;
    xAborted:=1;
    //xResetRequest:=(xExecute=0);
    xAgain:=0;(* !!! *)
END_IF
END_METHOD

{attribute 'hide' := ''}
METHOD PRIVATE FINAL HandleAbortingState
VAR_INPUT
END_VAR
VAR_OUTPUT
	xAgain: BOOL;
END_VAR
VAR
	xComplete: BOOL;
END_VAR
AbortAction(xComplete=> xComplete);

IF eErrorID<>Modbus_ErrorCode.NO_ERROR THEN
    eState:=STATE.INERROR;
    xAgain:=1;
ELSIF xComplete THEN
    eState:=STATE.ABORTED;
    xAgain:=1;
END_IF
END_METHOD

{attribute 'hide' := ''}
METHOD PRIVATE FINAL  HandleDoneState
VAR_OUTPUT
	xAgain: BOOL;
END_VAR
//在运行过程中要是切换模式，再运行完成之后，检测到模式的切换，就需要回到初始位置，进行下一次执行准备
IF _xDone AND xExecute=0 THEN
	eState:=STATE.RESETING;
	xAgain:=1;
ELSE
	xBusy:=0;
	_xDone:=1;
	//xResetRequest:=(xExecute=0);
	xAgain:=0;(* !!! *)
	IF _xDone AND xExecute AND NOT xOpe THEN
		xExecute:=0;
	END_IF	
END_IF
END_METHOD

{attribute 'hide' := ''}
METHOD PRIVATE FINAL  HandleDormantState
VAR_OUTPUT
	xAgain: BOOL;
END_VAR
IF xExecute THEN
    xBusy:=1;
    eState:=STATE.EXECUTING;
    xAgain:=1;
END_IF

//读取线圈,01
	IF stOpera.xReadCoilStatus
	THEN
		eCmd := Modbus_Cmd.ReadCoilStatus;
		xExecute := TRUE;
	END_IF

//读取输入线圈,02
	IF stOpera.xReadInputStatus
	THEN
		eCmd := Modbus_Cmd.ReadInputStatus;
		xExecute := TRUE;
	END_IF
	
//读取保持寄存器,03
	IF stOpera.xReadHoldingRegisters
	THEN
		eCmd := Modbus_Cmd.ReadHoldingRegisters;
		xExecute := TRUE;
	END_IF	

//读取输入寄存器,04
	IF stOpera.xReadInputRegisters
	THEN
		eCmd := Modbus_Cmd.ReadInputRegisters;
		xExecute := TRUE;
	END_IF
		
//写入单个线圈,05
	IF stOpera.xSetSingalCoil
	THEN
		eCmd := Modbus_Cmd.SetSingalCoil;
		xExecute := TRUE;
	END_IF
	
//写入单个保持寄存器,06
	IF stOpera.xSetSingalHoldingRegister
	THEN
		eCmd := Modbus_Cmd.SetSingalHoldingRegister;
		xExecute := TRUE;
	END_IF

//写入多个线圈,15
	IF stOpera.xSetMultiCoil
	THEN
		eCmd := Modbus_Cmd.SetMultiCoil;
		xExecute := TRUE;
	END_IF
	
//写入多个保持寄存器,16
	IF stOpera.xSetMultiHoldingRegister
	THEN
		eCmd := Modbus_Cmd.SetMultiHoldingRegister;
		xExecute := TRUE;
	END_IF
END_METHOD

{attribute 'hide' := ''}
METHOD PRIVATE FINAL  HandleErrorState
VAR_OUTPUT
	xAgain: BOOL;
END_VAR
IF xError AND  (xResetRequest OR NOT xExecute) THEN
    eState:=STATE.RESETING;
    xAgain:=1;
ELSE
    xBusy:=0;
    xError:=1;    
    xAgain:=0;(* !!! *)
END_IF
END_METHOD

{attribute 'hide' := ''}
METHOD PRIVATE FINAL  HandleExecutingState
VAR_OUTPUT
	xAgain: BOOL;
END_VAR
VAR
	xComplete: BOOL;
END_VAR

IF xAbort=0 THEN   
    CyclicAction(xComplete=> xComplete);
END_IF

IF eErrorID<>Modbus_ErrorCode.NO_ERROR THEN
    eState:=STATE.INERROR;
    xAgain:=1;
ELSIF xAbort THEN
    eState:=STATE.ABORTING;
    xAgain:=1;
ELSIF xComplete THEN
    eState:=STATE.DONE;
    xAgain:=1;
END_IF
END_METHOD

{attribute 'hide' := ''}
METHOD  PRIVATE FINAL  HandleResettingState
VAR_OUTPUT
	xAgain: BOOL;
END_VAR
VAR
	xComplete: BOOL;
END_VAR
ResetAction(xComplete=> xComplete);

IF xComplete THEN
		xExecute:=0;//清除输入指令 
    xBusy:=0;
    _xDone:=0;
    xError:=0;

    eErrorID:=Modbus_ErrorCode.NO_ERROR;
	eTCPErrorID := 0;
    eState:=STATE.DORMANT;
    xFirstInvocation:=1;//保证初始化信号
    xAgain:=0;(* !!! *)
END_IF
END_METHOD

{attribute 'hide' := ''}
METHOD PROTECTED ResetAction
VAR_OUTPUT
	xComplete: BOOL;
END_VAR
(*
* Cleaning
* => free all allocated resources
* => reinitialize instance variables
*)
tOperationTimer(IN:=0);
_tDelay(IN:=FALSE);
_tonTimeout(IN:= FALSE);
_xDone	:=FALSE;
_iSendNGCount := 0;
_fbTcpIpClient(xEnable:=FALSE);//将tcpip功能初始化、
sModbusError:='';
xComplete:=1;	
//复位操作标志
stOpera.xReadCoilStatus:=
stOpera.xReadHoldingRegisters:=
stOpera.xReadInputRegisters:=
stOpera.xReadInputStatus:=
stOpera.xSetMultiCoil:=
stOpera.xSetMultiHoldingRegister:=
stOpera.xSetSingalCoil:=
stOpera.xSetSingalHoldingRegister:=FALSE;
END_METHOD

END_FUNCTION_BLOCK

// ---- POUs/003_FB/53_RudongPump/41 Modbus指令/DataExchange/ModbusTCP_ErrorQuery.TcPOU
FUNCTION ModbusTCP_ErrorQuery : STRING
VAR_INPUT
	///错误编号
	ModbusTCP_ErrorNum: BYTE;
END_VAR

CASE ModbusTCP_ErrorNum OF
	16#00://	
(*
无错误
*)
		ModbusTCP_ErrorQuery:='Modbus_No_Error';
		
(*
非法功能，
对于服务器（或从站）来说，询问中接收到的功能码是不可允许的操作，
可能是因为功能码仅适用于新设备而被选单元中不可实现同时，
还指出服务器（或从站）在错误状态中处理这种请求，
例如：它是未配置的，且要求返回寄存器值 。
*)				
	16#01://
		ModbusTCP_ErrorQuery:='Modbus_IllegalFunction_Error';
		
(*
非法数据地址
对于服务器（或从站）来说，询问中接收的数据地址是不可允许的地址，
特别是参考号和传输长度的组合是无效的。对于带有100个寄存器的控制器来说，
偏移量96和长度4的请求会成功，而偏移量96和长度5的请求将产生异常码02。
*)		
	16#02://
		ModbusTCP_ErrorQuery:='Modbus_IllegalDataAddress_Error';
		
(*
非法数据值
对于服务器（或从站）来说，询问中包括的值是不可允许的值。该值指示了组合请求剩余结构中的故障。
例如：隐含长度是不正确的。modbus协议不知道任何特殊寄存器的任何特殊值的重要意义，
寄存器中被提交存储的数据项有一个应用程序期望之外的值。
*)					
	16#03://
		ModbusTCP_ErrorQuery:='Modbus_IllegalDataValue_Error';
		
(*
从站设备故障
当服务器（或从站）正在设法执行请求的操作时，产生不可重新获得的差错。
*)		
	16#04://
		ModbusTCP_ErrorQuery:='Modbus_SlaveBrakeDown_Error';
		
(*
确认与编程命令一起使用，服务器（或从站）已经接受请求，
并且正在处理这个请求，但是需要长持续时间进行这些操作，
返回这个响应防止在客户机（或主站）中发生超时错误，
客户机（或主机）可以继续发送轮询程序完成报文来确认是否完成处理。
*)				
	16#05://
		ModbusTCP_ErrorQuery:='Modbus_SlaveProcessing_Alarm';//指令正在处理	

(*
从属设备忙与编程命令一起使用，服务器（或从站）正在处理长持续时间的程序命令，
当服务器（或从站）空闲时，客户机（或主站）应该稍后重新传输报文。
*)		
	16#06://
		ModbusTCP_ErrorQuery:='Modbus_SlaveBusy_Error';	

(*
存储奇偶性差错与功能码20和21以及参考类型6一起使用，
指示扩展文件区不能通过一致性校验。服务器（或从站）设备读取记录文件，
但在存储器中发现一个奇偶校验错误。客户机（或主机）可重新发送请求，但可以在服务器（或从站）设备上要求服务。
*)		
	16#08://
		ModbusTCP_ErrorQuery:='Modbus_Parity_Error';	//校验错误，MODBUSTCP无此错误	
		
(*
不可用网关路径与网关一起使用，
指示网关不能为处理请求分配输入端口值输出端口的内部通信路径，
通常意味着网关是错误配置的或过载的。
*)		
	16#0A://
		ModbusTCP_ErrorQuery:='Modbus_GateWay_Error';	
		
(*
网关目标设备响应失败与网关一起使用，
指示没有从目标设备中获得响应，通常意味着设备未在网络中。
*)		
	16#0B://
		ModbusTCP_ErrorQuery:='Modbus_SlaveNon-existent';			
		
	ELSE
		ModbusTCP_ErrorQuery:='Modbus_SlaveNon-existent';
END_CASE

END_FUNCTION

// ---- POUs/003_FB/0000_FB_Alive/FB_Alive.TcPOU
FUNCTION_BLOCK FB_Alive
(*
********************************************************************************
* Name: FB_Alive
*
* Author:  AutomanH
* Version: 1.0.0
*
* Description:
* PLC and PC and Camera Communication Alive
*
* Remarks:
*
*  Revisions:
*   V1.0.0 -Automanh 2022.05.20
*********************************************************************************)
VAR_INPUT
iAliveSingle:INT;
END_VAR
VAR_OUTPUT
 xQAlive:BOOL;
 xQAliveError:BOOL;
END_VAR
VAR
tTonOff1s:TON;
tTonOn1s:TON;
tTimeOut:ARRAY[1..2] OF TON;
END_VAR

(* 	clock 1 second *)
tTonOff1s(IN:=NOT(tTonOn1s.Q),PT:=t#1s);
tTonOn1s(IN:=(tTonOff1s.Q),PT:=t#1s);

(* Live Bit *)
xQAlive := tTonOff1s.Q;

(*检测是否跳变**)
tTimeOut[1](IN:=(iAliveSingle =1),PT:=T#5S); 
tTimeOut[2](IN:=(iAliveSingle =0),PT:=T#5S); 
xQAliveError:=tTimeOut[1].Q OR tTimeOut[2].Q;

END_FUNCTION_BLOCK

// ---- POUs/003_FB/0009_MKC204C/FB_MKC204C.TcPOU
FUNCTION_BLOCK FB_MKC204C
(*
********************************************************************************
* Name: FB_MT_MKC_New
*
* Author:  Automanh
* Version: 1.0.0
*
* Description:
*  Re-Write  function block
*
* Remarks:
*
* Revisions:
*   1.0 -AutomanH Rebuild
		1.1- AutomanH 2022.07.27 add Error  FLT_CannotExecutable
														 add Excute Reset Command
*         
*  
*********************************************************************************)
VAR_INPUT
	
	xIReset:						BOOL	:= FALSE;		
	xIInit:  						BOOL ;
	iICodeLEN:					INT:=20;
	iICodePOS:					INT:=1;
	xIDeviceRunning			:BOOL;
	xManualMode					:BOOL;
	xAutoMode						:BOOL;
	stDeviceOpe					:ST_DeviceOpe;//秤体操作
	stpar								:ST_MCK_ParIn;
	stSysPar						:ST_SysPar;
END_VAR
VAR_OUTPUT
	xQRdyCmd:  						BOOL ;
	xQDone     :  				BOOL ;
	strQBarCode  : 				STRING[255];
	xQBusy:							BOOL	:= FALSE;	
	xQError:						BOOL	:= FALSE;	
  xQNoRead:					BOOL	:= FALSE;
	iQErrorNo:				INT;
	stParOut					: ST_MCK_ParOut;//参数输出
END_VAR
VAR_IN_OUT
	
END_VAR

VAR
 		{attribute 'tc_no_symbol'}
    	Waittime           :  TON ;
			{attribute 'tc_no_symbol'}
  		TcpIpClient  :  FB_LocalClient  ;
			{attribute 'tc_no_symbol'}
  		ClientSendBuffer  : ARRAY [1..80] OF BYTE ;
			{attribute 'tc_no_symbol'}
  		ClientRecvBuffer  : ARRAY [1..80] OF BYTE ;
			{attribute 'tc_no_symbol'}
			First  :  BOOL ;
			{attribute 'tc_no_symbol'}
    	strRead    :  STRING[10]    ;
			{attribute 'tc_no_symbol'}
    	strStop    :  STRING[5]  := 'LOFF$R'  ;
			{attribute 'tc_no_symbol'}
    	strBload    :  STRING[8] ;
			{attribute 'tc_no_symbol'}
    	eStepCmd	: E_ClientSteps ;
			{attribute 'tc_no_symbol'}
			strRecv : STRING[40] ;
			{attribute 'tc_no_symbol'}
			Done  : BOOL ;
			iStep     :  INT ;
			strLocalQBarCode  : 				STRING[255];
			iLoadStep: INT;
			xBloadStart: BOOL;
			strBloadResultCode:STRING(20);
			fbTrigger: R_TRIG;
			iCmdStep:INT;
			iCmdOldStep:INT;
			tTimeout:TON;
			eErrorID		: MT_MCK_ERROR;(*错误码*)(* Output: Error ID (defined below) *)
			xStart: BOOL ;
			xBusy:BOOL;
			xDone:BOOL;
			xRdyCmd:	BOOL ;
			xCmd:BOOL;
			OperR_TRIG:ARRAY[1..20] OF R_TRIG;
			i:INT;
	// //操作类型
		iOperType: INT;
		_Stemp: ARRAY[1..2] OF STRING[50];
			_sSendData: STRING(255);
			rTareSet: REAL;
	// 重复接收
	xRepeatReceive: BOOL;
END_VAR

VAR CONSTANT
	iMAX_LENGTH     :  INT := 255 ;
END_VAR

ACT_Op();
ACT_Cmd();
ACT_Reset();
ACT_Error();
ACT_RW();

ACTION ACT_Cmd:
IF  NOT  xQBusy THEN
 		xQRdyCmd:=TRUE;
ELSE
 		xQRdyCmd:=FALSE;	
END_IF
tTimeout(IN:= (iCmdStep =iCmdOldStep) AND (iCmdStep<>0)  AND (iOperType<>14), PT:= T#10S, Q=> , ET=> );
IF		tTimeout.Q THEN
 	xQError:=TRUE;
	eErrorID:=MT_MCK_ERROR.FLT_CMD_TIMEOUT;
END_IF
CASE iCmdStep  OF	
		
